C05480=1150.541,191.261,-61.437,-178.171,7.215,148.820
C05481=1150.545,191.011,-61.414,-178.174,7.213,148.820
C05482=1150.550,190.763,-61.390,-178.176,7.211,148.820
C05483=1150.554,190.514,-61.366,-178.180,7.208,148.820
C05484=1150.559,190.265,-61.343,-178.182,7.206,148.821
C05485=1150.564,190.016,-61.319,-178.185,7.203,148.821
C05486=1150.568,189.768,-61.295,-178.187,7.201,148.821
C05487=1150.573,189.519,-61.272,-178.191,7.199,148.821
C05488=1150.578,189.270,-61.249,-178.193,7.197,148.822
C05489=1150.582,189.020,-61.225,-178.196,7.194,148.822
C05490=1150.587,188.771,-61.202,-178.199,7.192,148.822
C05491=1150.591,188.523,-61.178,-178.202,7.189,148.822
C05492=1150.596,188.274,-61.155,-178.204,7.188,148.823
C05493=1150.601,188.025,-61.131,-178.208,7.185,148.823
C05494=1150.605,187.776,-61.108,-178.210,7.183,148.823
C05495=1150.609,187.527,-61.085,-178.213,7.181,148.823
C05496=1150.615,187.279,-61.062,-178.215,7.178,148.824
C05497=1150.619,187.030,-61.038,-178.218,7.177,148.824
C05498=1150.624,186.781,-61.015,-178.221,7.174,148.824
C05499=1150.628,186.532,-60.991,-178.224,7.172,148.824
C05500=1150.633,186.283,-60.968,-178.227,7.169,148.825
C05501=1150.637,186.035,-60.945,-178.229,7.167,148.825
C05502=1150.642,185.786,-60.922,-178.232,7.165,148.825
C05503=1150.647,185.537,-60.898,-178.235,7.163,148.826
C05504=1150.651,185.288,-60.875,-178.238,7.160,148.826
C05505=1150.656,185.039,-60.852,-178.240,7.158,148.826
C05506=1150.660,184.790,-60.829,-178.243,7.157,148.826
C05507=1150.665,184.541,-60.806,-178.246,7.154,148.827
C05508=1150.670,184.292,-60.783,-178.249,7.152,148.827
C05509=1150.675,184.023,-60.758,-178.252,7.149,148.827
C05510=1150.680,183.753,-60.733,-178.255,7.147,148.827
C05511=1150.684,183.483,-60.707,-178.257,7.145,148.828
C05512=1150.690,183.214,-60.682,-178.261,7.142,148.828
C05513=1150.694,182.965,-60.659,-178.264,7.140,148.828
C05514=1150.699,182.717,-60.636,-178.266,7.138,148.829
C05515=1150.704,182.467,-60.614,-178.269,7.136,148.829
C05516=1150.708,182.218,-60.590,-178.272,7.133,148.829
C05517=1150.712,181.969,-60.567,-178.274,7.131,148.829
C05518=1150.717,181.720,-60.544,-178.278,7.129,148.830
C05519=1150.722,181.471,-60.521,-178.280,7.127,148.830
C05520=1150.726,181.223,-60.498,-178.283,7.125,148.830
C05521=1150.731,180.973,-60.476,-178.286,7.122,148.831
C05522=1150.736,180.724,-60.452,-178.288,7.120,148.831
C05523=1150.740,180.476,-60.430,-178.291,7.118,148.831
C05524=1150.745,180.227,-60.406,-178.294,7.116,148.831
C05525=1150.749,179.979,-60.384,-178.297,7.113,148.832
C05526=1150.754,179.729,-60.361,-178.300,7.111,148.832
C05527=1150.759,179.480,-60.338,-178.302,7.109,148.832
C05528=1150.763,179.231,-60.315,-178.306,7.107,148.833
C05529=1150.768,178.983,-60.292,-178.308,7.105,148.833
C05530=1150.773,178.734,-60.270,-178.310,7.103,148.833
C05531=1150.777,178.484,-60.247,-178.314,7.101,148.833
C05532=1150.782,178.235,-60.223,-178.316,7.098,148.834
C05533=1150.787,177.987,-60.202,-178.319,7.096,148.834
C05534=1150.792,177.738,-60.178,-178.322,7.094,148.834
C05535=1150.796,177.489,-60.155,-178.324,7.092,148.834
C05536=1150.801,177.239,-60.133,-178.327,7.089,148.835
C05537=1150.805,176.991,-60.110,-178.330,7.088,148.835
C05538=1150.810,176.742,-60.087,-178.333,7.085,148.835
C05539=1150.814,176.493,-60.065,-178.336,7.083,148.836
C05540=1150.819,176.244,-60.042,-178.338,7.081,148.836
C05541=1150.824,175.995,-60.020,-178.342,7.079,148.836
C05542=1150.828,175.746,-59.997,-178.344,7.077,148.837
C05543=1150.833,175.497,-59.975,-178.346,7.075,148.837
C05544=1150.838,175.249,-59.952,-178.350,7.072,148.837
C05545=1150.842,174.999,-59.930,-178.352,7.070,148.837
C05546=1150.847,174.750,-59.906,-178.355,7.069,148.838
C05547=1150.852,174.502,-59.884,-178.358,7.066,148.838
C05548=1150.856,174.253,-59.862,-178.361,7.064,148.838
C05549=1150.861,174.003,-59.839,-178.363,7.061,148.839
C05550=1150.865,173.755,-59.817,-178.366,7.060,148.839
C05551=1150.870,173.506,-59.794,-178.369,7.058,148.839
C05552=1150.874,173.257,-59.771,-178.372,7.055,148.839
C05553=1150.880,173.008,-59.749,-178.374,7.053,148.840
C05554=1150.884,172.759,-59.726,-178.377,7.052,148.840
C05555=1150.889,172.511,-59.705,-178.380,7.049,148.841
C05556=1150.894,172.261,-59.682,-178.383,7.047,148.841
C05557=1150.898,172.012,-59.659,-178.385,7.045,148.841
C05558=1150.902,171.764,-59.637,-178.389,7.043,148.841
C05559=1150.907,171.515,-59.614,-178.391,7.041,148.842
C05560=1150.911,171.265,-59.592,-178.393,7.039,148.842
C05561=1150.916,171.017,-59.570,-178.397,7.036,148.842
C05562=1150.921,170.767,-59.547,-178.399,7.035,148.843
C05563=1150.926,170.519,-59.525,-178.402,7.033,148.843
C05564=1150.930,170.270,-59.503,-178.405,7.030,148.843
C05565=1150.936,170.021,-59.481,-178.408,7.028,148.843
C05566=1150.940,169.772,-59.458,-178.410,7.026,148.844
C05567=1150.944,169.522,-59.436,-178.414,7.024,148.844
C05568=1150.950,169.274,-59.414,-178.416,7.022,148.844
C05569=1150.954,169.024,-59.392,-178.419,7.020,148.845
C05570=1150.958,168.776,-59.369,-178.422,7.017,148.845
C05571=1150.963,168.527,-59.347,-178.425,7.016,148.845
C05572=1150.968,168.278,-59.325,-178.427,7.014,148.846
C05573=1150.973,168.029,-59.303,-178.430,7.011,148.846
C05574=1150.977,167.780,-59.281,-178.433,7.009,148.846
C05575=1150.981,167.531,-59.259,-178.435,7.008,148.847
C05576=1150.987,167.282,-59.236,-178.438,7.006,148.847
C05577=1150.991,167.033,-59.214,-178.441,7.003,148.847
C05578=1150.996,166.784,-59.192,-178.444,7.001,148.848
C05579=1151.000,166.535,-59.171,-178.446,7.000,148.848
C05580=1151.005,166.286,-59.149,-178.450,6.997,148.848
C05581=1151.010,166.037,-59.126,-178.452,6.995,148.848
C05582=1151.015,165.788,-59.105,-178.455,6.993,148.849
C05583=1151.019,165.539,-59.082,-178.457,6.991,148.849
C05584=1151.024,165.291,-59.060,-178.461,6.989,148.850
C05585=1151.028,165.041,-59.038,-178.463,6.987,148.850
C05586=1151.033,164.793,-59.016,-178.465,6.985,148.850
C05587=1151.037,164.543,-58.994,-178.469,6.983,148.850
C05588=1151.043,164.294,-58.972,-178.471,6.981,148.851
C05589=1151.047,164.045,-58.950,-178.474,6.979,148.851
C05590=1151.052,163.796,-58.928,-178.477,6.977,148.852
C05591=1151.056,163.547,-58.906,-178.480,6.974,148.852
C05592=1151.061,163.298,-58.885,-178.482,6.973,148.852
C05593=1151.066,163.049,-58.863,-178.485,6.971,148.852
C05594=1151.070,162.800,-58.841,-178.488,6.968,148.853
C05595=1151.075,162.551,-58.819,-178.491,6.967,148.853
C05596=1151.080,162.302,-58.798,-178.493,6.965,148.853
C05597=1151.085,162.053,-58.776,-178.496,6.963,148.854
C05598=1151.089,161.804,-58.754,-178.499,6.960,148.854
C05599=1151.094,161.555,-58.732,-178.502,6.959,148.854
C05600=1151.098,161.306,-58.710,-178.505,6.957,148.855
C05601=1151.103,161.057,-58.689,-178.507,6.955,148.855
C05602=1151.108,160.809,-58.667,-178.510,6.952,148.855
C05603=1151.112,160.559,-58.645,-178.513,6.951,148.856
C05604=1151.117,160.310,-58.624,-178.516,6.949,148.856
C05605=1151.122,160.061,-58.602,-178.518,6.947,148.856
C05606=1151.126,159.812,-58.580,-178.522,6.945,148.857
C05607=1151.131,159.563,-58.559,-178.524,6.943,148.857
C05608=1151.136,159.314,-58.537,-178.526,6.941,148.857
C05609=1151.141,159.065,-58.516,-178.529,6.939,148.858
C05610=1151.146,158.816,-58.494,-178.532,6.936,148.858
C05611=1151.150,158.567,-58.472,-178.535,6.935,148.858
C05612=1151.155,158.318,-58.450,-178.538,6.933,148.859
C05613=1151.160,158.049,-58.427,-178.541,6.930,148.859
C05614=1151.165,157.780,-58.404,-178.544,6.929,148.860
C05615=1151.170,157.511,-58.381,-178.547,6.926,148.860
C05616=1151.175,157.242,-58.357,-178.550,6.924,148.860
C05617=1151.180,156.993,-58.336,-178.553,6.923,148.861
C05618=1151.185,156.744,-58.315,-178.555,6.921,148.861
C05619=1151.189,156.495,-58.293,-178.558,6.918,148.861
C05620=1151.194,156.246,-58.272,-178.561,6.916,148.862
C05621=1151.199,155.997,-58.250,-178.563,6.915,148.862
C05622=1151.203,155.748,-58.228,-178.566,6.913,148.862
C05623=1151.208,155.498,-58.207,-178.569,6.910,148.863
C05624=1151.213,155.250,-58.186,-178.572,6.909,148.863
C05625=1151.218,155.001,-58.165,-178.575,6.907,148.863
C05626=1151.222,154.752,-58.143,-178.577,6.905,148.864
C05627=1151.226,154.503,-58.122,-178.580,6.903,148.864
C05628=1151.232,154.254,-58.101,-178.583,6.901,148.864
C05629=1151.236,154.005,-58.079,-178.586,6.899,148.865
C05630=1151.241,153.755,-58.058,-178.589,6.897,148.865
C05631=1151.245,153.507,-58.037,-178.591,6.895,148.865
C05632=1151.250,153.257,-58.016,-178.594,6.894,148.866
C05633=1151.255,153.009,-57.994,-178.597,6.891,148.866
C05634=1151.260,152.759,-57.973,-178.600,6.889,148.867
C05635=1151.264,152.511,-57.952,-178.602,6.887,148.867
C05636=1151.269,152.261,-57.931,-178.605,6.886,148.867
C05637=1151.274,152.012,-57.910,-178.608,6.884,148.868
C05638=1151.279,151.763,-57.888,-178.611,6.881,148.868
C05639=1151.283,151.514,-57.867,-178.614,6.880,148.868
C05640=1151.288,151.265,-57.846,-178.616,6.878,148.869
C05641=1151.293,151.016,-57.825,-178.619,6.876,148.869
C05642=1151.298,150.767,-57.804,-178.622,6.874,148.869
C05643=1151.302,150.518,-57.782,-178.624,6.873,148.870
C05644=1151.307,150.268,-57.761,-178.628,6.870,148.870
C05645=1151.312,150.019,-57.740,-178.630,6.868,148.870
C05646=1151.316,149.771,-57.719,-178.633,6.866,148.871
C05647=1151.321,149.521,-57.698,-178.635,6.865,148.871
C05648=1151.327,149.272,-57.677,-178.638,6.863,148.871
C05649=1151.331,149.024,-57.656,-178.641,6.861,148.872
C05650=1151.335,148.774,-57.635,-178.644,6.859,148.872
C05651=1151.340,148.525,-57.614,-178.647,6.857,148.873
C05652=1151.345,148.276,-57.593,-178.649,6.855,148.873
C05653=1151.350,148.027,-57.572,-178.652,6.854,148.873
C05654=1151.354,147.778,-57.551,-178.655,6.852,148.874
C05655=1151.359,147.529,-57.530,-178.658,6.850,148.874
C05656=1151.364,147.280,-57.510,-178.661,6.848,148.875
C05657=1151.368,147.031,-57.488,-178.664,6.846,148.875
C05658=1151.373,146.781,-57.467,-178.666,6.844,148.875
C05659=1151.378,146.532,-57.447,-178.668,6.842,148.875
C05660=1151.383,146.283,-57.426,-178.671,6.840,148.876
C05661=1151.387,146.034,-57.405,-178.674,6.839,148.876
C05662=1151.392,145.785,-57.384,-178.677,6.837,148.877
C05663=1151.397,145.537,-57.363,-178.680,6.834,148.877
C05664=1151.402,145.287,-57.342,-178.683,6.833,148.877
C05665=1151.406,145.038,-57.322,-178.685,6.831,148.878
C05666=1151.411,144.789,-57.301,-178.688,6.829,148.878
C05667=1151.416,144.540,-57.281,-178.691,6.827,148.879
C05668=1151.421,144.291,-57.260,-178.693,6.826,148.879
C05669=1151.425,144.041,-57.239,-178.696,6.824,148.879
C05670=1151.430,143.792,-57.218,-178.699,6.822,148.880
C05671=1151.434,143.543,-57.198,-178.702,6.820,148.880
C05672=1151.440,143.294,-57.177,-178.705,6.818,148.880
C05673=1151.444,143.045,-57.156,-178.708,6.816,148.881
C05674=1151.449,142.796,-57.134,-178.710,6.815,148.881
C05675=1151.453,142.547,-57.114,-178.713,6.813,148.882
C05676=1151.458,142.298,-57.094,-178.716,6.811,148.882
C05677=1151.463,142.048,-57.073,-178.718,6.809,148.882
C05678=1151.468,141.799,-57.053,-178.721,6.808,148.883
C05679=1151.473,141.550,-57.032,-178.723,6.806,148.883
C05680=1151.477,141.301,-57.012,-178.727,6.803,148.883
C05681=1151.482,141.052,-56.991,-178.729,6.801,148.884
C05682=1151.487,140.803,-56.970,-178.732,6.800,148.884
C05683=1151.491,140.554,-56.950,-178.735,6.798,148.884
C05684=1151.496,140.305,-56.930,-178.737,6.796,148.885
C05685=1151.501,140.056,-56.909,-178.740,6.795,148.885
C05686=1151.505,139.807,-56.888,-178.743,6.793,148.886
C05687=1151.511,139.558,-56.867,-178.746,6.791,148.886
C05688=1151.515,139.309,-56.847,-178.748,6.789,148.886
C05689=1151.520,139.059,-56.827,-178.751,6.788,148.887
C05690=1151.525,138.810,-56.806,-178.754,6.785,148.887
C05691=1151.529,138.561,-56.786,-178.757,6.783,148.888
C05692=1151.534,138.312,-56.766,-178.760,6.782,148.888
C05693=1151.539,138.064,-56.746,-178.762,6.780,148.888
C05694=1151.544,137.814,-56.725,-178.765,6.778,148.889
C05695=1151.549,137.565,-56.705,-178.768,6.777,148.889
C05696=1151.553,137.316,-56.685,-178.771,6.775,148.890
C05697=1151.558,137.067,-56.664,-178.773,6.773,148.890
C05698=1151.563,136.817,-56.644,-178.776,6.771,148.890
C05699=1151.568,136.568,-56.624,-178.779,6.770,148.891
C05700=1151.572,136.319,-56.603,-178.781,6.768,148.891
C05701=1151.577,136.070,-56.582,-178.784,6.766,148.891
C05702=1151.582,135.820,-56.563,-178.787,6.765,148.892
C05703=1151.586,135.571,-56.542,-178.790,6.763,148.892
C05704=1151.591,135.323,-56.522,-178.793,6.760,148.893
C05705=1151.596,135.074,-56.503,-178.796,6.759,148.893
C05706=1151.601,134.824,-56.482,-178.798,6.757,148.893
C05707=1151.606,134.575,-56.461,-178.801,6.755,148.894
C05708=1151.611,134.326,-56.442,-178.804,6.753,148.894
C05709=1151.615,134.077,-56.421,-178.806,6.752,148.895
C05710=1151.620,133.827,-56.402,-178.809,6.750,148.895
C05711=1151.624,133.578,-56.381,-178.812,6.748,148.895
C05712=1151.630,133.330,-56.361,-178.815,6.747,148.896
C05713=1151.635,133.080,-56.341,-178.818,6.745,148.896
C05714=1151.639,132.831,-56.321,-178.821,6.744,148.897
C05715=1151.644,132.582,-56.301,-178.823,6.742,148.897
C05716=1151.648,132.333,-56.281,-178.826,6.740,148.898
C05717=1151.654,132.064,-56.259,-178.829,6.738,148.898
C05718=1151.659,131.796,-56.237,-178.832,6.736,148.898
C05719=1151.664,131.527,-56.215,-178.835,6.734,148.899
C05720=1151.669,131.258,-56.194,-178.837,6.732,148.899
C05721=1151.674,131.010,-56.174,-178.840,6.731,148.900
C05722=1151.679,130.760,-56.155,-178.843,6.729,148.900
C05723=1151.683,130.511,-56.134,-178.846,6.728,148.901
C05724=1151.688,130.262,-56.115,-178.849,6.726,148.901
C05725=1151.693,130.012,-56.095,-178.851,6.724,148.901
C05726=1151.698,129.764,-56.075,-178.854,6.723,148.902
C05727=1151.703,129.514,-56.055,-178.857,6.721,148.902
C05728=1151.707,129.266,-56.035,-178.860,6.719,148.903
C05729=1151.712,129.016,-56.015,-178.862,6.717,148.903
C05730=1151.717,128.767,-55.996,-178.865,6.716,148.903
C05731=1151.722,128.518,-55.975,-178.868,6.714,148.904
C05732=1151.727,128.268,-55.955,-178.870,6.712,148.904
C05733=1151.731,128.019,-55.935,-178.873,6.711,148.904
C05734=1151.736,127.771,-55.916,-178.876,6.709,148.905
C05735=1151.741,127.521,-55.897,-178.879,6.707,148.905
C05736=1151.745,127.272,-55.876,-178.881,6.705,148.906
C05737=1151.751,127.023,-55.857,-178.884,6.704,148.906
C05738=1151.755,126.774,-55.837,-178.887,6.702,148.906
C05739=1151.760,126.524,-55.818,-178.889,6.700,148.907
C05740=1151.765,126.275,-55.797,-178.893,6.699,148.908
C05741=1151.770,126.026,-55.778,-178.895,6.697,148.908
C05742=1151.775,125.777,-55.758,-178.898,6.696,148.908
C05743=1151.779,125.527,-55.739,-178.901,6.694,148.909
C05744=1151.784,125.279,-55.719,-178.904,6.692,148.909
C05745=1151.789,125.029,-55.699,-178.906,6.690,148.909
C05746=1151.794,124.780,-55.679,-178.909,6.689,148.910
C05747=1151.799,124.531,-55.660,-178.912,6.687,148.910
C05748=1151.803,124.282,-55.641,-178.914,6.685,148.911
C05749=1151.808,124.033,-55.621,-178.917,6.684,148.911
C05750=1151.812,123.783,-55.601,-178.920,6.682,148.911
C05751=1151.818,123.534,-55.582,-178.923,6.680,148.912
C05752=1151.822,123.285,-55.562,-178.926,6.679,148.913
C05753=1151.828,123.036,-55.543,-178.928,6.677,148.913
C05754=1151.832,122.787,-55.524,-178.931,6.675,148.913
C05755=1151.837,122.537,-55.504,-178.934,6.674,148.914
C05756=1151.842,122.289,-55.484,-178.937,6.672,148.914
C05757=1151.846,122.039,-55.464,-178.939,6.670,148.915
C05758=1151.851,121.790,-55.445,-178.942,6.669,148.915
C05759=1151.856,121.541,-55.425,-178.945,6.667,148.915
C05760=1151.860,121.292,-55.406,-178.947,6.665,148.916
C05761=1151.866,121.043,-55.387,-178.950,6.663,148.916
C05762=1151.871,120.793,-55.367,-178.953,6.662,148.917
C05763=1151.875,120.544,-55.348,-178.956,6.660,148.917
C05764=1151.880,120.295,-55.329,-178.959,6.659,148.918
C05765=1151.885,120.045,-55.309,-178.962,6.657,148.918
C05766=1151.890,119.797,-55.290,-178.964,6.655,148.918
C05767=1151.895,119.547,-55.270,-178.967,6.654,148.919
C05768=1151.899,119.298,-55.251,-178.969,6.653,148.919
C05769=1151.904,119.049,-55.232,-178.972,6.651,148.920
C05770=1151.909,118.799,-55.212,-178.975,6.649,148.920
C05771=1151.913,118.551,-55.194,-178.978,6.648,148.921
C05772=1151.918,118.301,-55.174,-178.980,6.646,148.921
C05773=1151.923,118.052,-55.155,-178.983,6.645,148.921
C05774=1151.929,117.802,-55.136,-178.986,6.643,148.922
C05775=1151.933,117.554,-55.117,-178.989,6.641,148.922
C05776=1151.938,117.304,-55.098,-178.991,6.639,148.923
C05777=1151.943,117.055,-55.078,-178.994,6.638,148.923
C05778=1151.947,116.806,-55.059,-178.997,6.636,148.923
C05779=1151.952,116.556,-55.040,-179.000,6.635,148.924
C05780=1151.957,116.307,-55.020,-179.003,6.633,148.924
C05781=1151.962,116.058,-55.002,-179.005,6.631,148.925
C05782=1151.967,115.809,-54.983,-179.008,6.630,148.925
C05783=1151.971,115.559,-54.964,-179.010,6.629,148.926
C05784=1151.976,115.311,-54.944,-179.013,6.627,148.926
C05785=1151.981,115.061,-54.925,-179.016,6.625,148.926
C05786=1151.986,114.812,-54.907,-179.018,6.624,148.927
C05787=1151.991,114.563,-54.887,-179.022,6.622,148.927
C05788=1151.995,114.314,-54.868,-179.024,6.621,148.928
C05789=1152.001,114.065,-54.849,-179.027,6.619,148.928
C05790=1152.006,113.815,-54.830,-179.030,6.617,148.929
C05791=1152.010,113.566,-54.811,-179.033,6.615,148.929
C05792=1152.015,113.317,-54.792,-179.035,6.615,148.930
C05793=1152.020,113.067,-54.774,-179.038,6.613,148.930
C05794=1152.025,112.818,-54.754,-179.041,6.612,148.931
C05795=1152.029,112.569,-54.735,-179.043,6.610,148.931
C05796=1152.034,112.319,-54.716,-179.046,6.608,148.931
C05797=1152.039,112.071,-54.698,-179.049,6.606,148.932
C05798=1152.044,111.822,-54.678,-179.052,6.605,148.932
C05799=1152.049,111.572,-54.660,-179.054,6.603,148.933
C05800=1152.054,111.323,-54.641,-179.057,6.602,148.933
C05801=1152.058,111.074,-54.622,-179.060,6.601,148.934
C05802=1152.064,110.824,-54.603,-179.062,6.599,148.934
C05803=1152.068,110.576,-54.584,-179.065,6.597,148.934
C05804=1152.073,110.325,-54.566,-179.068,6.596,148.935
C05805=1152.078,110.077,-54.547,-179.070,6.594,148.935
C05806=1152.083,109.827,-54.528,-179.074,6.593,148.936
C05807=1152.088,109.578,-54.509,-179.076,6.591,148.936
C05808=1152.093,109.329,-54.491,-179.079,6.589,148.937
C05809=1152.097,109.079,-54.472,-179.081,6.588,148.937
C05810=1152.102,108.831,-54.453,-179.084,6.587,148.938
C05811=1152.107,108.581,-54.434,-179.087,6.585,148.938
C05812=1152.112,108.331,-54.416,-179.090,6.584,148.939
C05813=1152.117,108.083,-54.397,-179.093,6.582,148.939
C05814=1152.121,107.833,-54.378,-179.095,6.580,148.939
C05815=1152.126,107.584,-54.360,-179.098,6.579,148.940
C05816=1152.132,107.335,-54.341,-179.100,6.578,148.940
C05817=1152.136,107.085,-54.322,-179.103,6.576,148.941
C05818=1152.141,106.836,-54.303,-179.106,6.575,148.941
C05819=1152.146,106.587,-54.285,-179.109,6.573,148.942
C05820=1152.150,106.337,-54.266,-179.112,6.571,148.942
C05821=1152.156,106.069,-54.246,-179.114,6.570,148.943
C05822=1152.161,105.801,-54.226,-179.118,6.568,148.943
C05823=1152.167,105.533,-54.206,-179.120,6.567,148.944
C05824=1152.171,105.264,-54.186,-179.123,6.565,148.944
C05825=1152.176,105.015,-54.168,-179.126,6.564,148.945
C05826=1152.181,104.766,-54.149,-179.129,6.562,148.945
C05827=1152.186,104.517,-54.131,-179.132,6.560,148.945
C05828=1152.191,104.267,-54.113,-179.134,6.559,148.946
C05829=1152.196,104.018,-54.094,-179.137,6.558,148.946
C05830=1152.201,103.769,-54.076,-179.140,6.556,148.947
C05831=1152.205,103.519,-54.057,-179.142,6.555,148.947
C05832=1152.210,103.270,-54.039,-179.145,6.553,148.948
C05833=1152.215,103.021,-54.020,-179.147,6.552,148.948
C05834=1152.220,102.772,-54.002,-179.151,6.551,148.949
C05835=1152.225,102.522,-53.984,-179.153,6.549,148.949
C05836=1152.229,102.273,-53.965,-179.156,6.547,148.950
C05837=1152.235,102.024,-53.946,-179.159,6.546,148.950
C05838=1152.240,101.774,-53.928,-179.161,6.544,148.950
C05839=1152.245,101.525,-53.910,-179.164,6.543,148.951
C05840=1152.249,101.275,-53.892,-179.167,6.542,148.951
C05841=1152.254,101.027,-53.873,-179.170,6.540,148.952
C05842=1152.259,100.777,-53.855,-179.172,6.538,148.952
C05843=1152.264,100.528,-53.837,-179.175,6.537,148.953
C05844=1152.269,100.278,-53.818,-179.178,6.536,148.953
C05845=1152.273,100.029,-53.800,-179.180,6.534,148.954
C05846=1152.278,99.780,-53.783,-179.183,6.533,148.954
C05847=1152.283,99.531,-53.765,-179.186,6.531,148.955
C05848=1152.289,99.282,-53.745,-179.189,6.530,148.955
C05849=1152.293,99.032,-53.727,-179.191,6.529,148.956
C05850=1152.298,98.783,-53.709,-179.194,6.527,148.956
C05851=1152.303,98.534,-53.691,-179.197,6.525,148.956
C05852=1152.308,98.285,-53.673,-179.200,6.524,148.957
C05853=1152.313,98.035,-53.655,-179.203,6.522,148.958
C05854=1152.318,97.786,-53.637,-179.205,6.522,148.958
C05855=1152.322,97.536,-53.619,-179.207,6.520,148.958
C05856=1152.327,97.287,-53.601,-179.210,6.518,148.959
C05857=1152.332,97.038,-53.582,-179.213,6.517,148.959
C05858=1152.337,96.788,-53.564,-179.215,6.516,148.960
C05859=1152.342,96.539,-53.546,-179.218,6.514,148.960
C05860=1152.347,96.290,-53.528,-179.221,6.513,148.961
C05861=1152.352,96.041,-53.510,-179.224,6.511,148.961
C05862=1152.356,95.791,-53.492,-179.226,6.510,148.962
C05863=1152.361,95.542,-53.474,-179.229,6.509,148.962
C05864=1152.366,95.293,-53.456,-179.232,6.507,148.963
C05865=1152.371,95.044,-53.438,-179.235,6.506,148.963
C05866=1152.376,94.794,-53.420,-179.238,6.504,148.964
C05867=1152.381,94.545,-53.402,-179.240,6.503,148.964
C05868=1152.386,94.295,-53.385,-179.243,6.501,148.964
C05869=1152.391,94.046,-53.367,-179.246,6.500,148.965
C05870=1152.396,93.797,-53.349,-179.249,6.498,148.966
C05871=1152.401,93.548,-53.331,-179.251,6.498,148.966
C05872=1152.405,93.298,-53.312,-179.253,6.496,148.966
C05873=1152.410,93.049,-53.294,-179.257,6.495,148.967
C05874=1152.415,92.800,-53.276,-179.259,6.493,148.967
C05875=1152.420,92.550,-53.259,-179.261,6.492,148.968
C05876=1152.425,92.301,-53.241,-179.264,6.490,148.968
C05877=1152.430,92.051,-53.223,-179.267,6.489,148.969
C05878=1152.435,91.802,-53.205,-179.270,6.487,148.969
C05879=1152.439,91.553,-53.188,-179.272,6.486,148.970
C05880=1152.444,91.304,-53.171,-179.275,6.485,148.970
C05881=1152.449,91.054,-53.153,-179.278,6.483,148.971
C05882=1152.454,90.805,-53.135,-179.280,6.483,148.971
C05883=1152.459,90.556,-53.117,-179.283,6.481,148.972
C05884=1152.464,90.306,-53.099,-179.286,6.480,148.972
C05885=1152.469,90.057,-53.081,-179.289,6.478,148.973
C05886=1152.474,89.808,-53.063,-179.291,6.477,148.973
C05887=1152.479,89.559,-53.045,-179.294,6.475,148.974
C05888=1152.484,89.309,-53.029,-179.297,6.474,148.974
C05889=1152.488,89.060,-53.011,-179.300,6.472,148.975
C05890=1152.493,88.811,-52.993,-179.302,6.471,148.975
C05891=1152.499,88.561,-52.976,-179.305,6.470,148.975
C05892=1152.503,88.312,-52.958,-179.308,6.468,148.976
C05893=1152.508,88.063,-52.940,-179.310,6.468,148.977
C05894=1152.513,87.813,-52.923,-179.313,6.466,148.977
C05895=1152.518,87.564,-52.905,-179.316,6.465,148.978
C05896=1152.523,87.314,-52.888,-179.319,6.463,148.978
C05897=1152.528,87.065,-52.870,-179.321,6.462,148.978
C05898=1152.533,86.816,-52.852,-179.324,6.460,148.979
C05899=1152.537,86.567,-52.835,-179.327,6.459,148.980
C05900=1152.542,86.317,-52.817,-179.329,6.458,148.980
C05901=1152.547,86.068,-52.800,-179.332,6.456,148.980
C05902=1152.552,85.818,-52.782,-179.335,6.455,148.981
C05903=1152.557,85.569,-52.765,-179.337,6.454,148.981
C05904=1152.562,85.320,-52.747,-179.340,6.453,148.982
C05905=1152.567,85.070,-52.730,-179.343,6.451,148.982
C05906=1152.572,84.821,-52.712,-179.346,6.450,148.983
C05907=1152.577,84.572,-52.696,-179.348,6.449,148.983
C05908=1152.582,84.323,-52.678,-179.351,6.447,148.984
C05909=1152.587,84.073,-52.660,-179.354,6.446,148.984
C05910=1152.591,83.824,-52.643,-179.356,6.445,148.985
C05911=1152.596,83.574,-52.626,-179.359,6.443,148.985
C05912=1152.601,83.325,-52.608,-179.362,6.442,148.986
C05913=1152.606,83.076,-52.591,-179.364,6.441,148.986
C05914=1152.611,82.826,-52.573,-179.367,6.439,148.987
C05915=1152.616,82.577,-52.556,-179.370,6.438,148.987
C05916=1152.621,82.328,-52.540,-179.372,6.437,148.988
C05917=1152.626,82.079,-52.522,-179.375,6.435,148.988
C05918=1152.631,81.829,-52.504,-179.378,6.434,148.989
C05919=1152.635,81.580,-52.487,-179.380,6.433,148.989
C05920=1152.641,81.330,-52.470,-179.383,6.432,148.990
C05921=1152.646,81.080,-52.452,-179.386,6.430,148.990
C05922=1152.650,80.832,-52.435,-179.388,6.429,148.991
C05923=1152.656,80.583,-52.418,-179.391,6.428,148.991
C05924=1152.660,80.333,-52.401,-179.394,6.426,148.992
C05925=1152.666,80.064,-52.383,-179.397,6.426,148.992
C05926=1152.671,79.796,-52.363,-179.399,6.424,148.993
C05927=1152.676,79.528,-52.346,-179.403,6.423,148.993
C05928=1152.681,79.259,-52.327,-179.405,6.421,148.994
C05929=1152.687,79.009,-52.310,-179.408,6.420,148.995
C05930=1152.692,78.761,-52.293,-179.411,6.419,148.995
C05931=1152.697,78.511,-52.275,-179.413,6.417,148.995
C05932=1152.701,78.262,-52.259,-179.417,6.416,148.996
C05933=1152.706,78.012,-52.241,-179.419,6.415,148.996
C05934=1152.711,77.763,-52.225,-179.421,6.413,148.997
C05935=1152.716,77.514,-52.207,-179.424,6.411,148.997
C05936=1152.721,77.265,-52.190,-179.427,6.411,148.998
C05937=1152.726,77.015,-52.173,-179.430,6.409,148.998
C05938=1152.730,76.765,-52.157,-179.432,6.408,148.999
C05939=1152.736,76.516,-52.139,-179.435,6.407,149.000
C05940=1152.741,76.267,-52.123,-179.438,6.405,149.000
C05941=1152.746,76.018,-52.105,-179.440,6.405,149.000
C05942=1152.750,75.768,-52.088,-179.443,6.403,149.001
C05943=1152.755,75.518,-52.071,-179.446,6.402,149.001
C05944=1152.760,75.270,-52.055,-179.448,6.401,149.002
C05945=1152.766,75.020,-52.037,-179.451,6.399,149.003
C05946=1152.770,74.770,-52.021,-179.453,6.399,149.003
C05947=1152.775,74.521,-52.004,-179.456,6.397,149.003
C05948=1152.780,74.272,-51.987,-179.459,6.396,149.004
C05949=1152.786,74.022,-51.970,-179.461,6.395,149.004
C05950=1152.790,73.772,-51.953,-179.464,6.393,149.005
C05951=1152.795,73.524,-51.936,-179.467,6.393,149.006
C05952=1152.800,73.275,-51.919,-179.470,6.391,149.006
C05953=1152.805,73.025,-51.902,-179.472,6.389,149.006
C05954=1152.810,72.775,-51.885,-179.475,6.389,149.007
C05955=1152.815,72.526,-51.869,-179.478,6.387,149.008
C05956=1152.819,72.277,-51.852,-179.480,6.387,149.008
C05957=1152.825,72.027,-51.835,-179.483,6.385,149.009
C05958=1152.830,71.778,-51.819,-179.486,6.383,149.009
C05959=1152.834,71.529,-51.802,-179.488,6.383,149.010
C05960=1152.839,71.279,-51.785,-179.491,6.381,149.010
C05961=1152.845,71.030,-51.769,-179.493,6.380,149.011
C05962=1152.849,70.780,-51.752,-179.496,6.379,149.011
C05963=1152.854,70.530,-51.735,-179.499,6.377,149.012
C05964=1152.860,70.282,-51.719,-179.501,6.376,149.012
C05965=1152.864,70.032,-51.702,-179.505,6.375,149.013
C05966=1152.869,69.782,-51.685,-179.507,6.374,149.013
C05967=1152.874,69.534,-51.669,-179.509,6.372,149.014
C05968=1152.879,69.284,-51.652,-179.513,6.371,149.014
C05969=1152.884,69.034,-51.635,-179.515,6.370,149.015
C05970=1152.889,68.786,-51.618,-179.518,6.369,149.015
C05971=1152.894,68.535,-51.602,-179.520,6.368,149.016
C05972=1152.899,68.287,-51.586,-179.523,6.366,149.016
C05973=1152.904,68.037,-51.569,-179.526,6.366,149.017
C05974=1152.909,67.787,-51.552,-179.528,6.364,149.017
C05975=1152.914,67.539,-51.536,-179.531,6.363,149.018
C05976=1152.918,67.289,-51.519,-179.534,6.362,149.018
C05977=1152.924,67.039,-51.503,-179.536,6.361,149.019
C05978=1152.929,66.790,-51.486,-179.539,6.360,149.019
C05979=1152.933,66.540,-51.470,-179.542,6.358,149.020
C05980=1152.938,66.292,-51.453,-179.544,6.357,149.020
C05981=1152.944,66.041,-51.437,-179.547,6.356,149.021
C05982=1152.949,65.792,-51.420,-179.549,6.355,149.021
C05983=1152.954,65.543,-51.404,-179.552,6.354,149.022
C05984=1152.958,65.293,-51.387,-179.555,6.352,149.023
C05985=1152.963,65.044,-51.372,-179.557,6.352,149.023
C05986=1152.968,64.795,-51.355,-179.560,6.350,149.023
C05987=1152.974,64.545,-51.338,-179.563,6.349,149.024
C05988=1152.978,64.295,-51.322,-179.566,6.348,149.025
C05989=1152.984,64.047,-51.306,-179.568,6.347,149.025
C05990=1152.988,63.797,-51.289,-179.571,6.346,149.026
C05991=1152.993,63.548,-51.273,-179.573,6.345,149.026
C05992=1152.998,63.298,-51.257,-179.576,6.343,149.027
C05993=1153.003,63.049,-51.240,-179.579,6.343,149.027
C05994=1153.008,62.799,-51.224,-179.581,6.341,149.028
C05995=1153.013,62.550,-51.207,-179.585,6.340,149.028
C05996=1153.018,62.300,-51.192,-179.587,6.339,149.029
C05997=1153.023,62.051,-51.175,-179.589,6.337,149.029
C05998=1153.028,61.802,-51.159,-179.592,6.337,149.030
C05999=1153.033,61.552,-51.143,-179.595,6.335,149.030
C06000=1153.038,61.303,-51.126,-179.597,6.334,149.031
C06001=1153.043,61.053,-51.110,-179.600,6.333,149.031
C06002=1153.048,60.804,-51.094,-179.602,6.332,149.032
C06003=1153.052,60.554,-51.078,-179.606,6.331,149.032
C06004=1153.058,60.305,-51.062,-179.608,6.330,149.033
C06005=1153.063,60.056,-51.046,-179.611,6.328,149.034
C06006=1153.067,59.806,-51.030,-179.613,6.328,149.034
C06007=1153.072,59.558,-51.013,-179.616,6.326,149.034
C06008=1153.077,59.307,-50.997,-179.618,6.325,149.035
C06009=1153.083,59.058,-50.981,-179.621,6.324,149.036
C06010=1153.088,58.808,-50.965,-179.624,6.323,149.036
C06011=1153.093,58.559,-50.949,-179.627,6.322,149.037
C06012=1153.098,58.309,-50.932,-179.629,6.321,149.037
C06013=1153.103,58.060,-50.917,-179.632,6.319,149.038
C06014=1153.108,57.811,-50.900,-179.634,6.319,149.038
C06015=1153.112,57.561,-50.885,-179.637,6.317,149.039
C06016=1153.117,57.313,-50.869,-179.640,6.316,149.039
C06017=1153.122,57.062,-50.853,-179.642,6.315,149.040
C06018=1153.127,56.813,-50.837,-179.645,6.314,149.040
C06019=1153.132,56.564,-50.821,-179.648,6.313,149.041
C06020=1153.137,56.314,-50.805,-179.650,6.312,149.041
C06021=1153.143,56.065,-50.789,-179.653,6.311,149.042
C06022=1153.147,55.815,-50.773,-179.655,6.310,149.042
C06023=1153.153,55.566,-50.757,-179.658,6.308,149.043
C06024=1153.157,55.316,-50.741,-179.661,6.308,149.043
C06025=1153.162,55.067,-50.725,-179.664,6.306,149.044
C06026=1153.168,54.818,-50.709,-179.666,6.305,149.045
C06027=1153.173,54.568,-50.693,-179.669,6.304,149.045
C06028=1153.178,54.319,-50.677,-179.671,6.303,149.046
C06029=1153.183,54.050,-50.660,-179.674,6.302,149.046
C06030=1153.189,53.782,-50.643,-179.677,6.301,149.047
C06031=1153.193,53.513,-50.626,-179.680,6.300,149.047
C06032=1153.199,53.244,-50.609,-179.683,6.298,149.048
C06033=1153.204,52.995,-50.594,-179.685,6.298,149.049
C06034=1153.209,52.745,-50.578,-179.688,6.296,149.049
C06035=1153.214,52.496,-50.562,-179.690,6.295,149.049
C06036=1153.219,52.247,-50.546,-179.693,6.294,149.050
C06037=1153.224,51.997,-50.530,-179.696,6.293,149.051
C06038=1153.229,51.748,-50.515,-179.699,6.292,149.051
C06039=1153.234,51.498,-50.499,-179.701,6.291,149.052
C06040=1153.239,51.248,-50.483,-179.704,6.289,149.052
C06041=1153.244,50.999,-50.467,-179.706,6.289,149.053
C06042=1153.249,50.750,-50.451,-179.709,6.288,149.053
C06043=1153.254,50.501,-50.436,-179.712,6.287,149.054
C06044=1153.259,50.251,-50.420,-179.714,6.286,149.054
C06045=1153.264,50.001,-50.405,-179.717,6.284,149.055
C06046=1153.270,49.752,-50.389,-179.719,6.284,149.055
C06047=1153.274,49.502,-50.373,-179.722,6.282,149.056
C06048=1153.279,49.253,-50.358,-179.725,6.281,149.057
C06049=1153.284,49.004,-50.342,-179.727,6.280,149.057
C06050=1153.289,48.754,-50.326,-179.730,6.279,149.058
C06051=1153.293,48.505,-50.311,-179.732,6.278,149.058
C06052=1153.299,48.255,-50.295,-179.735,6.277,149.059
C06053=1153.304,48.006,-50.280,-179.738,6.276,149.059
C06054=1153.309,47.756,-50.264,-179.740,6.275,149.060
C06055=1153.314,47.507,-50.249,-179.743,6.274,149.060
C06056=1153.319,47.257,-50.233,-179.746,6.273,149.061
C06057=1153.324,47.008,-50.218,-179.748,6.272,149.061
C06058=1153.329,46.758,-50.202,-179.751,6.271,149.062
C06059=1153.334,46.509,-50.187,-179.753,6.270,149.062
C06060=1153.339,46.259,-50.171,-179.756,6.269,149.063
C06061=1153.344,46.010,-50.156,-179.759,6.267,149.063
C06062=1153.349,45.761,-50.141,-179.761,6.267,149.064
C06063=1153.354,45.511,-50.125,-179.764,6.265,149.065
C06064=1153.359,45.262,-50.110,-179.767,6.265,149.065
C06065=1153.364,45.012,-50.094,-179.769,6.264,149.066
C06066=1153.370,44.763,-50.079,-179.772,6.262,149.066
C06067=1153.374,44.513,-50.063,-179.774,6.262,149.067
C06068=1153.379,44.264,-50.048,-179.777,6.260,149.067
C06069=1153.384,44.014,-50.032,-179.780,6.260,149.068
C06070=1153.389,43.764,-50.018,-179.782,6.259,149.068
C06071=1153.395,43.515,-50.002,-179.785,6.258,149.069
C06072=1153.399,43.266,-49.987,-179.787,6.257,149.069
C06073=1153.404,43.016,-49.971,-179.790,6.255,149.070
C06074=1153.410,42.766,-49.956,-179.793,6.255,149.071
C06075=1153.414,42.517,-49.941,-179.795,6.254,149.071
C06076=1153.420,42.268,-49.925,-179.798,6.253,149.072
C06077=1153.425,42.018,-49.911,-179.800,6.252,149.072
C06078=1153.430,41.769,-49.895,-179.803,6.250,149.073
C06079=1153.434,41.519,-49.880,-179.806,6.250,149.073
C06080=1153.439,41.270,-49.864,-179.808,6.249,149.074
C06081=1153.445,41.020,-49.849,-179.811,6.247,149.074
C06082=1153.450,40.771,-49.834,-179.813,6.247,149.075
C06083=1153.455,40.521,-49.819,-179.816,6.245,149.075
C06084=1153.460,40.272,-49.804,-179.819,6.244,149.076
C06085=1153.465,40.023,-49.788,-179.821,6.244,149.077
C06086=1153.470,39.773,-49.774,-179.824,6.242,149.077
C06087=1153.475,39.523,-49.758,-179.827,6.242,149.078
C06088=1153.479,39.274,-49.743,-179.829,6.241,149.078
C06089=1153.485,39.024,-49.727,-179.832,6.240,149.079
C06090=1153.490,38.775,-49.713,-179.834,6.239,149.079
C06091=1153.495,38.525,-49.697,-179.837,6.237,149.080
C06092=1153.500,38.276,-49.682,-179.840,6.237,149.080
C06093=1153.506,38.026,-49.668,-179.842,6.236,149.081
C06094=1153.510,37.777,-49.653,-179.845,6.235,149.082
C06095=1153.515,37.528,-49.638,-179.847,6.234,149.082
C06096=1153.521,37.278,-49.623,-179.850,6.233,149.083
C06097=1153.525,37.029,-49.608,-179.853,6.232,149.083
C06098=1153.531,36.779,-49.592,-179.855,6.231,149.084
C06099=1153.535,36.529,-49.578,-179.857,6.230,149.084
C06100=1153.540,36.280,-49.562,-179.860,6.229,149.085
C06101=1153.545,36.031,-49.547,-179.863,6.228,149.085
C06102=1153.550,35.781,-49.533,-179.865,6.227,149.086
C06103=1153.555,35.531,-49.517,-179.868,6.226,149.086
C06104=1153.560,35.282,-49.503,-179.870,6.225,149.087
C06105=1153.566,35.032,-49.487,-179.874,6.224,149.088
C06106=1153.571,34.783,-49.473,-179.876,6.223,149.088
C06107=1153.575,34.533,-49.458,-179.878,6.223,149.089
C06108=1153.581,34.283,-49.443,-179.881,6.221,149.089
C06109=1153.586,34.034,-49.428,-179.884,6.221,149.090
C06110=1153.591,33.785,-49.412,-179.886,6.220,149.090
C06111=1153.596,33.535,-49.398,-179.889,6.219,149.091
C06112=1153.601,33.286,-49.383,-179.891,6.218,149.091
C06113=1153.606,33.036,-49.368,-179.893,6.217,149.092
C06114=1153.611,32.787,-49.353,-179.897,6.216,149.093
C06115=1153.616,32.537,-49.339,-179.899,6.215,149.093
C06116=1153.621,32.288,-49.323,-179.902,6.214,149.094
C06117=1153.626,32.038,-49.309,-179.904,6.213,149.094
C06118=1153.631,31.789,-49.295,-179.907,6.212,149.095
C06119=1153.636,31.539,-49.280,-179.909,6.211,149.095
C06120=1153.642,31.289,-49.265,-179.912,6.210,149.096
C06121=1153.646,31.040,-49.250,-179.915,6.209,149.096
C06122=1153.651,30.791,-49.236,-179.917,6.209,149.097
C06123=1153.657,30.541,-49.220,-179.920,6.207,149.098
C06124=1153.661,30.292,-49.206,-179.923,6.207,149.098
C06125=1153.666,30.042,-49.192,-179.925,6.206,149.099
C06126=1153.671,29.793,-49.177,-179.927,6.205,149.099
C06127=1153.677,29.543,-49.162,-179.930,6.204,149.100
C06128=1153.682,29.294,-49.148,-179.932,6.203,149.100
C06129=1153.687,29.045,-49.133,-179.935,6.202,149.101
C06130=1153.692,28.795,-49.119,-179.938,6.201,149.101
C06131=1153.697,28.545,-49.104,-179.940,6.200,149.102
C06132=1153.702,28.296,-49.089,-179.943,6.200,149.103
C06133=1153.707,28.027,-49.073,-179.946,6.198,149.103
C06134=1153.713,27.758,-49.058,-179.948,6.198,149.104
C06135=1153.719,27.488,-49.042,-179.951,6.196,149.104
C06136=1153.724,27.220,-49.026,-179.954,6.196,149.105
C06137=1153.729,26.970,-49.012,-179.956,6.195,149.105
C06138=1153.733,26.721,-48.997,-179.959,6.194,149.106
C06139=1153.739,26.472,-48.983,-179.961,6.193,149.107
C06140=1153.745,26.222,-48.968,-179.964,6.192,149.107
C06141=1153.750,25.972,-48.954,-179.967,6.191,149.108
C06142=1153.754,25.723,-48.939,-179.969,6.190,149.108
C06143=1153.759,25.473,-48.924,-179.972,6.189,149.109
C06144=1153.764,25.224,-48.910,-179.975,6.188,149.110
C06145=1153.769,24.974,-48.896,-179.977,6.187,149.110
C06146=1153.774,24.724,-48.882,-179.980,6.187,149.111
C06147=1153.780,24.475,-48.866,-179.982,6.186,149.111
C06148=1153.785,24.226,-48.852,-179.985,6.185,149.112
C06149=1153.790,23.976,-48.838,-179.987,6.184,149.112
C06150=1153.795,23.726,-48.824,-179.989,6.183,149.113
C06151=1153.800,23.477,-48.809,-179.992,6.183,149.113
C06152=1153.805,23.227,-48.795,-179.995,6.181,149.114
C06153=1153.810,22.978,-48.780,-179.997,6.180,149.115
C06154=1153.815,22.729,-48.766,-180.000,6.180,149.115
C06155=1153.820,22.479,-48.752,179.997,6.178,149.116
C06156=1153.825,22.229,-48.738,179.995,6.178,149.116
C06157=1153.830,21.980,-48.723,179.992,6.177,149.117
C06158=1153.835,21.730,-48.709,179.990,6.176,149.117
C06159=1153.840,21.481,-48.695,179.987,6.175,149.118
C06160=1153.845,21.231,-48.681,179.985,6.174,149.118
C06161=1153.850,20.982,-48.667,179.982,6.174,149.119
C06162=1153.855,20.732,-48.652,179.980,6.173,149.120
C06163=1153.860,20.482,-48.638,179.977,6.172,149.120
C06164=1153.867,20.233,-48.623,179.975,6.171,149.121
C06165=1153.872,19.983,-48.609,179.972,6.170,149.121
C06166=1153.876,19.733,-48.595,179.970,6.169,149.122
C06167=1153.881,19.484,-48.581,179.966,6.168,149.122
C06168=1153.886,19.234,-48.567,179.964,6.167,149.123
C06169=1153.891,18.985,-48.553,179.962,6.167,149.124
C06170=1153.896,18.736,-48.539,179.959,6.166,149.124
C06171=1153.901,18.486,-48.524,179.956,6.165,149.125
C06172=1153.906,18.236,-48.510,179.954,6.164,149.125
C06173=1153.912,17.987,-48.496,179.951,6.164,149.126
C06174=1153.917,17.737,-48.482,179.949,6.163,149.126
C06175=1153.922,17.488,-48.468,179.946,6.161,149.127
C06176=1153.926,17.238,-48.453,179.944,6.161,149.127
C06177=1153.932,16.989,-48.440,179.942,6.160,149.128
C06178=1153.937,16.739,-48.425,179.939,6.159,149.129
C06179=1153.942,16.490,-48.411,179.937,6.159,149.129
C06180=1153.948,16.241,-48.397,179.934,6.157,149.130
C06181=1153.952,15.991,-48.383,179.931,6.156,149.130
C06182=1153.958,15.741,-48.369,179.929,6.156,149.131
C06183=1153.963,15.491,-48.355,179.927,6.155,149.131
C06184=1153.967,15.242,-48.342,179.923,6.154,149.132
C06185=1153.972,14.992,-48.327,179.921,6.153,149.133
C06186=1153.977,14.743,-48.313,179.919,6.153,149.133
C06187=1153.983,14.494,-48.299,179.916,6.152,149.134
C06188=1153.988,14.244,-48.285,179.914,6.151,149.134
C06189=1153.993,13.994,-48.271,179.911,6.150,149.135
C06190=1153.999,13.745,-48.257,179.908,6.149,149.135
C06191=1154.003,13.495,-48.244,179.906,6.148,149.136
C06192=1154.008,13.246,-48.229,179.903,6.148,149.137
C06193=1154.013,12.997,-48.216,179.901,6.147,149.137
C06194=1154.019,12.746,-48.202,179.898,6.146,149.138
C06195=1154.024,12.496,-48.188,179.896,6.145,149.138
C06196=1154.029,12.247,-48.174,179.893,6.145,149.139
C06197=1154.033,11.998,-48.160,179.891,6.144,149.139
C06198=1154.039,11.748,-48.147,179.888,6.143,149.140
C06199=1154.044,11.499,-48.133,179.886,6.142,149.141
C06200=1154.049,11.249,-48.118,179.883,6.141,149.141
C06201=1154.054,10.999,-48.105,179.881,6.140,149.142
C06202=1154.059,10.750,-48.092,179.878,6.140,149.142
C06203=1154.064,10.500,-48.077,179.876,6.139,149.143
C06204=1154.070,10.251,-48.063,179.873,6.138,149.143
C06205=1154.075,10.001,-48.050,179.871,6.137,149.144
C06206=1154.079,9.752,-48.036,179.868,6.137,149.145
C06207=1154.085,9.503,-48.022,179.866,6.136,149.145
C06208=1154.090,9.252,-48.009,179.863,6.135,149.146
C06209=1154.095,9.002,-47.994,179.860,6.134,149.146
C06210=1154.100,8.753,-47.982,179.858,6.133,149.147
C06211=1154.105,8.503,-47.967,179.856,6.133,149.147
C06212=1154.111,8.254,-47.954,179.853,6.132,149.148
C06213=1154.115,8.004,-47.941,179.851,6.131,149.149
C06214=1154.121,7.755,-47.927,179.848,6.131,149.149
C06215=1154.126,7.505,-47.913,179.845,6.129,149.150
C06216=1154.131,7.255,-47.899,179.843,6.129,149.150
C06217=1154.136,7.007,-47.885,179.840,6.128,149.151
C06218=1154.141,6.756,-47.872,179.838,6.127,149.152
C06219=1154.147,6.507,-47.858,179.836,6.127,149.152
C06220=1154.151,6.257,-47.845,179.833,6.126,149.153
C06221=1154.157,6.008,-47.831,179.830,6.125,149.153
C06222=1154.162,5.758,-47.818,179.828,6.124,149.154
C06223=1154.166,5.509,-47.804,179.825,6.123,149.154
C06224=1154.172,5.259,-47.791,179.823,6.123,149.155
C06225=1154.176,5.010,-47.777,179.821,6.122,149.155
C06226=1154.182,4.760,-47.764,179.818,6.121,149.156
C06227=1154.187,4.510,-47.750,179.815,6.120,149.157
C06228=1154.192,4.261,-47.737,179.813,6.119,149.157
C06229=1154.197,4.011,-47.723,179.810,6.119,149.158
C06230=1154.203,3.762,-47.709,179.808,6.118,149.158
C06231=1154.207,3.512,-47.696,179.805,6.117,149.159
C06232=1154.213,3.263,-47.683,179.803,6.117,149.159
C06233=1154.217,3.013,-47.669,179.801,6.116,149.160
C06234=1154.223,2.764,-47.656,179.798,6.115,149.160
C06235=1154.228,2.513,-47.643,179.795,6.114,149.161
C06236=1154.233,2.264,-47.629,179.793,6.113,149.162
C06237=1154.239,1.994,-47.615,179.790,6.113,149.162
C06238=1154.244,1.725,-47.600,179.788,6.112,149.163
C06239=1154.250,1.457,-47.586,179.784,6.111,149.164
C06240=1154.255,1.187,-47.571,179.782,6.110,149.164
C06241=1154.260,0.937,-47.558,179.780,6.110,149.165
C06242=1154.266,0.688,-47.544,179.777,6.109,149.165
C06243=1154.271,0.437,-47.531,179.775,6.109,149.166
C06244=1154.276,0.189,-47.518,179.772,6.107,149.166
C06245=1154.281,-0.061,-47.504,179.769,6.107,149.167
C06246=1154.286,-0.311,-47.491,179.767,6.106,149.168
C06247=1154.292,-0.560,-47.477,179.765,6.105,149.168
C06248=1154.296,-0.810,-47.464,179.762,6.104,149.169
C06249=1154.302,-1.060,-47.451,179.760,6.104,149.169
C06250=1154.306,-1.310,-47.438,179.758,6.103,149.170
C06251=1154.312,-1.559,-47.424,179.755,6.103,149.171
C06252=1154.317,-1.809,-47.411,179.752,6.101,149.171
C06253=1154.322,-2.058,-47.398,179.749,6.101,149.172
C06254=1154.327,-2.307,-47.385,179.747,6.100,149.172
C06255=1154.332,-2.557,-47.372,179.745,6.099,149.173
C06256=1154.338,-2.807,-47.359,179.742,6.099,149.173
C06257=1154.342,-3.057,-47.346,179.740,6.098,149.174
C06258=1154.348,-3.306,-47.333,179.738,6.097,149.175
C06259=1154.353,-3.555,-47.319,179.735,6.097,149.175
C06260=1154.358,-3.805,-47.306,179.733,6.096,149.176
C06261=1154.363,-4.055,-47.293,179.730,6.095,149.176
C06262=1154.368,-4.305,-47.280,179.727,6.094,149.177
C06263=1154.374,-4.554,-47.267,179.725,6.094,149.178
C06264=1154.378,-4.803,-47.254,179.723,6.093,149.178
C06265=1154.384,-5.053,-47.240,179.720,6.092,149.179
C06266=1154.389,-5.303,-47.227,179.718,6.092,149.179
C06267=1154.394,-5.552,-47.215,179.715,6.091,149.180
C06268=1154.399,-5.802,-47.201,179.713,6.090,149.180
C06269=1154.404,-6.052,-47.189,179.710,6.090,149.181
C06270=1154.410,-6.302,-47.175,179.708,6.089,149.181
C06271=1154.414,-6.551,-47.162,179.705,6.089,149.182
C06272=1154.419,-6.800,-47.149,179.703,6.087,149.183
C06273=1154.425,-7.050,-47.136,179.700,6.087,149.183
C06274=1154.430,-7.300,-47.123,179.698,6.086,149.184
C06275=1154.435,-7.549,-47.110,179.695,6.085,149.184
C06276=1154.440,-7.799,-47.097,179.693,6.085,149.185
C06277=1154.445,-8.049,-47.084,179.690,6.084,149.186
C06278=1154.451,-8.298,-47.072,179.688,6.083,149.186
C06279=1154.455,-8.548,-47.059,179.685,6.083,149.187
C06280=1154.461,-8.798,-47.046,179.683,6.082,149.187
C06281=1154.466,-9.047,-47.033,179.681,6.082,149.188
C06282=1154.471,-9.297,-47.020,179.678,6.081,149.188
C06283=1154.476,-9.547,-47.007,179.676,6.080,149.189
C06284=1154.482,-9.796,-46.994,179.674,6.080,149.190
C06285=1154.487,-10.045,-46.982,179.670,6.078,149.190
C06286=1154.491,-10.295,-46.969,179.668,6.077,149.191
C06287=1154.497,-10.545,-46.955,179.666,6.077,149.191
C06288=1154.502,-10.794,-46.943,179.663,6.076,149.192
C06289=1154.507,-11.044,-46.930,179.661,6.076,149.193
C06290=1154.512,-11.294,-46.917,179.659,6.075,149.193
C06291=1154.518,-11.543,-46.904,179.656,6.075,149.194
C06292=1154.523,-11.793,-46.891,179.654,6.074,149.194
C06293=1154.527,-12.043,-46.878,179.651,6.073,149.195
C06294=1154.532,-12.292,-46.866,179.649,6.073,149.195
C06295=1154.538,-12.541,-46.853,179.646,6.072,149.196
C06296=1154.543,-12.791,-46.840,179.644,6.071,149.197
C06297=1154.548,-13.041,-46.828,179.641,6.071,149.197
C06298=1154.553,-13.291,-46.815,179.639,6.070,149.198
C06299=1154.558,-13.540,-46.803,179.637,6.070,149.198
C06300=1154.564,-13.790,-46.789,179.634,6.069,149.199
C06301=1154.569,-14.040,-46.776,179.632,6.068,149.200
C06302=1154.574,-14.289,-46.764,179.630,6.068,149.200
C06303=1154.579,-14.538,-46.751,179.627,6.067,149.201
C06304=1154.584,-14.788,-46.739,179.624,6.066,149.201
C06305=1154.589,-15.038,-46.726,179.621,6.065,149.202
C06306=1154.595,-15.288,-46.713,179.619,6.064,149.202
C06307=1154.600,-15.537,-46.701,179.617,6.064,149.203
C06308=1154.605,-15.787,-46.688,179.614,6.063,149.203
C06309=1154.610,-16.036,-46.675,179.612,6.063,149.204
C06310=1154.615,-16.287,-46.663,179.610,6.062,149.205
C06311=1154.620,-16.536,-46.651,179.607,6.061,149.205
C06312=1154.625,-16.785,-46.638,179.605,6.061,149.206
C06313=1154.631,-17.034,-46.625,179.602,6.060,149.207
C06314=1154.637,-17.285,-46.613,179.600,6.059,149.207
C06315=1154.641,-17.535,-46.600,179.597,6.059,149.208
C06316=1154.646,-17.784,-46.587,179.595,6.058,149.208
C06317=1154.651,-18.033,-46.575,179.592,6.058,149.209
C06318=1154.657,-18.283,-46.563,179.590,6.057,149.209
C06319=1154.662,-18.533,-46.550,179.588,6.056,149.210
C06320=1154.667,-18.782,-46.538,179.585,6.056,149.210
C06321=1154.672,-19.033,-46.525,179.583,6.055,149.211
C06322=1154.677,-19.282,-46.513,179.581,6.054,149.212
C06323=1154.682,-19.531,-46.500,179.578,6.054,149.212
C06324=1154.687,-19.781,-46.488,179.576,6.053,149.213
C06325=1154.693,-20.030,-46.476,179.573,6.053,149.214
C06326=1154.698,-20.280,-46.463,179.571,6.052,149.214
C06327=1154.703,-20.530,-46.451,179.568,6.051,149.215
C06328=1154.709,-20.779,-46.438,179.566,6.051,149.215
C06329=1154.714,-21.029,-46.425,179.563,6.050,149.216
C06330=1154.719,-21.279,-46.413,179.561,6.049,149.216
C06331=1154.724,-21.529,-46.401,179.559,6.049,149.217
C06332=1154.729,-21.778,-46.388,179.556,6.048,149.217
C06333=1154.735,-22.028,-46.376,179.554,6.048,149.218
C06334=1154.740,-22.277,-46.363,179.551,6.047,149.219
C06335=1154.745,-22.527,-46.352,179.549,6.047,149.219
C06336=1154.750,-22.776,-46.339,179.547,6.046,149.220
C06337=1154.756,-23.026,-46.326,179.544,6.045,149.220
C06338=1154.761,-23.276,-46.315,179.542,6.045,149.221
C06339=1154.766,-23.526,-46.302,179.539,6.044,149.222
C06340=1154.770,-23.775,-46.290,179.537,6.043,149.222
C06341=1154.777,-24.045,-46.276,179.534,6.043,149.223
C06342=1154.782,-24.315,-46.263,179.532,6.042,149.223
C06343=1154.787,-24.585,-46.250,179.529,6.042,149.224
C06344=1154.794,-24.855,-46.237,179.526,6.040,149.225
C06345=1154.798,-25.104,-46.225,179.525,6.040,149.225
C06346=1154.803,-25.354,-46.213,179.522,6.040,149.226
C06347=1154.809,-25.604,-46.201,179.520,6.039,149.226
C06348=1154.814,-25.853,-46.188,179.517,6.039,149.227
C06349=1154.819,-26.103,-46.176,179.515,6.038,149.228
C06350=1154.824,-26.353,-46.163,179.512,6.038,149.228
C06351=1154.829,-26.603,-46.151,179.510,6.037,149.229
C06352=1154.835,-26.853,-46.140,179.507,6.036,149.229
C06353=1154.840,-27.102,-46.127,179.505,6.036,149.230
C06354=1154.845,-27.352,-46.116,179.503,6.035,149.231
C06355=1154.850,-27.601,-46.103,179.500,6.034,149.231
C06356=1154.855,-27.851,-46.091,179.498,6.034,149.232
C06357=1154.860,-28.100,-46.079,179.496,6.033,149.232
C06358=1154.866,-28.350,-46.067,179.493,6.033,149.233
C06359=1154.871,-28.600,-46.055,179.491,6.032,149.233
C06360=1154.876,-28.849,-46.042,179.488,6.031,149.234
C06361=1154.881,-29.099,-46.031,179.486,6.031,149.235
C06362=1154.886,-29.349,-46.019,179.483,6.030,149.235
C06363=1154.891,-29.598,-46.006,179.481,6.029,149.236
C06364=1154.897,-29.848,-45.994,179.478,6.029,149.236
C06365=1154.902,-30.098,-45.982,179.476,6.028,149.237
C06366=1154.907,-30.347,-45.971,179.474,6.028,149.238
C06367=1154.912,-30.597,-45.959,179.471,6.027,149.238
C06368=1154.917,-30.846,-45.946,179.469,6.027,149.239
C06369=1154.923,-31.096,-45.934,179.466,6.026,149.239
C06370=1154.928,-31.346,-45.922,179.464,6.025,149.240
C06371=1154.933,-31.596,-45.911,179.462,6.025,149.240
C06372=1154.938,-31.845,-45.898,179.460,6.025,149.241
C06373=1154.943,-32.095,-45.887,179.457,6.024,149.242
C06374=1154.949,-32.344,-45.875,179.455,6.023,149.242
C06375=1154.954,-32.593,-45.863,179.453,6.023,149.243
C06376=1154.959,-32.843,-45.851,179.450,6.022,149.243
C06377=1154.965,-33.093,-45.839,179.448,6.022,149.244
C06378=1154.970,-33.343,-45.827,179.446,6.021,149.244
C06379=1154.975,-33.593,-45.816,179.443,6.020,149.245
C06380=1154.980,-33.842,-45.803,179.441,6.020,149.246
C06381=1154.985,-34.092,-45.792,179.438,6.019,149.246
C06382=1154.991,-34.342,-45.780,179.436,6.018,149.247
C06383=1154.995,-34.592,-45.768,179.433,6.018,149.247
C06384=1155.001,-34.841,-45.756,179.431,6.017,149.248
C06385=1155.006,-35.091,-45.744,179.429,6.018,149.249
C06386=1155.011,-35.341,-45.733,179.427,6.017,149.249
C06387=1155.016,-35.591,-45.721,179.424,6.016,149.250
C06388=1155.022,-35.840,-45.709,179.422,6.016,149.250
C06389=1155.028,-36.090,-45.697,179.419,6.015,149.251
C06390=1155.032,-36.339,-45.685,179.417,6.014,149.251
C06391=1155.037,-36.589,-45.673,179.414,6.014,149.252
C06392=1155.043,-36.839,-45.662,179.412,6.013,149.253
C06393=1155.047,-37.088,-45.650,179.410,6.013,149.253
C06394=1155.053,-37.338,-45.638,179.407,6.012,149.254
C06395=1155.058,-37.588,-45.627,179.405,6.012,149.254
C06396=1155.064,-37.837,-45.616,179.402,6.011,149.255
C06397=1155.069,-38.087,-45.604,179.400,6.011,149.256
C06398=1155.074,-38.337,-45.592,179.398,6.010,149.256
C06399=1155.079,-38.587,-45.581,179.396,6.010,149.257
C06400=1155.084,-38.836,-45.568,179.393,6.009,149.257
C06401=1155.089,-39.085,-45.557,179.391,6.008,149.258
C06402=1155.094,-39.335,-45.545,179.389,6.008,149.258
C06403=1155.100,-39.585,-45.533,179.386,6.007,149.259
C06404=1155.105,-39.834,-45.522,179.384,6.007,149.260
C06405=1155.111,-40.084,-45.510,179.381,6.006,149.260
C06406=1155.115,-40.334,-45.499,179.379,6.006,149.261
C06407=1155.121,-40.584,-45.487,179.377,6.006,149.261
C06408=1155.126,-40.834,-45.475,179.375,6.005,149.262
C06409=1155.131,-41.083,-45.464,179.372,6.004,149.262
C06410=1155.137,-41.333,-45.452,179.370,6.004,149.263
C06411=1155.142,-41.582,-45.441,179.368,6.003,149.264
C06412=1155.147,-41.832,-45.429,179.365,6.003,149.264
C06413=1155.152,-42.082,-45.418,179.363,6.002,149.265
C06414=1155.158,-42.331,-45.406,179.360,6.002,149.266
C06415=1155.162,-42.581,-45.395,179.358,6.001,149.266
C06416=1155.168,-42.831,-45.383,179.356,6.001,149.267
C06417=1155.173,-43.080,-45.372,179.354,6.000,149.267
C06418=1155.178,-43.331,-45.361,179.351,6.000,149.268
C06419=1155.184,-43.580,-45.350,179.349,5.999,149.268
C06420=1155.189,-43.830,-45.338,179.347,5.998,149.269
C06421=1155.194,-44.080,-45.326,179.344,5.998,149.270
C06422=1155.199,-44.329,-45.315,179.342,5.997,149.270
C06423=1155.204,-44.578,-45.304,179.339,5.997,149.271
C06424=1155.210,-44.828,-45.292,179.337,5.997,149.271
C06425=1155.215,-45.078,-45.281,179.335,5.996,149.272
C06426=1155.220,-45.328,-45.269,179.333,5.996,149.272
C06427=1155.225,-45.577,-45.257,179.330,5.995,149.273
C06428=1155.231,-45.827,-45.247,179.328,5.994,149.274
C06429=1155.236,-46.077,-45.235,179.325,5.994,149.274
C06430=1155.241,-46.327,-45.223,179.323,5.993,149.275
C06431=1155.246,-46.576,-45.212,179.321,5.994,149.275
C06432=1155.252,-46.825,-45.201,179.319,5.993,149.276
C06433=1155.257,-47.075,-45.189,179.316,5.992,149.276
C06434=1155.262,-47.326,-45.178,179.314,5.992,149.277
C06435=1155.268,-47.575,-45.167,179.312,5.991,149.278
C06436=1155.272,-47.824,-45.156,179.309,5.990,149.278
C06437=1155.278,-48.074,-45.144,179.307,5.990,149.279
C06438=1155.283,-48.324,-45.133,179.305,5.990,149.279
C06439=1155.289,-48.574,-45.122,179.302,5.989,149.280
C06440=1155.293,-48.823,-45.111,179.300,5.989,149.281
C06441=1155.298,-49.073,-45.099,179.298,5.988,149.281
C06442=1155.304,-49.322,-45.088,179.295,5.988,149.282
C06443=1155.309,-49.572,-45.077,179.293,5.987,149.282
C06444=1155.315,-49.822,-45.065,179.290,5.986,149.283
C06445=1155.321,-50.093,-45.053,179.288,5.986,149.283
C06446=1155.326,-50.363,-45.042,179.285,5.985,149.284
C06447=1155.331,-50.634,-45.030,179.283,5.984,149.285
C06448=1155.337,-50.904,-45.017,179.280,5.984,149.285
C06449=1155.342,-51.154,-45.006,179.278,5.984,149.286
C06450=1155.348,-51.404,-44.994,179.276,5.984,149.286
C06451=1155.353,-51.653,-44.984,179.273,5.983,149.287
C06452=1155.358,-51.903,-44.973,179.271,5.982,149.288
C06453=1155.363,-52.153,-44.961,179.269,5.982,149.288
C06454=1155.369,-52.402,-44.950,179.266,5.981,149.289
C06455=1155.374,-52.652,-44.940,179.265,5.981,149.289
C06456=1155.379,-52.902,-44.928,179.262,5.981,149.290
C06457=1155.384,-53.151,-44.917,179.260,5.980,149.291
C06458=1155.389,-53.401,-44.906,179.257,5.980,149.291
C06459=1155.395,-53.651,-44.895,179.255,5.979,149.292
C06460=1155.400,-53.901,-44.884,179.252,5.978,149.292
C06461=1155.405,-54.151,-44.873,179.251,5.978,149.293
C06462=1155.410,-54.399,-44.862,179.249,5.978,149.293
C06463=1155.416,-54.650,-44.851,179.246,5.977,149.294
C06464=1155.421,-54.900,-44.839,179.244,5.976,149.295
C06465=1155.426,-55.149,-44.829,179.241,5.976,149.295
C06466=1155.431,-55.399,-44.818,179.240,5.976,149.296
C06467=1155.437,-55.649,-44.807,179.237,5.976,149.296
C06468=1155.442,-55.898,-44.796,179.235,5.975,149.297
C06469=1155.447,-56.148,-44.785,179.232,5.974,149.298
C06470=1155.452,-56.397,-44.774,179.230,5.974,149.298
C06471=1155.458,-56.647,-44.762,179.228,5.974,149.299
C06472=1155.463,-56.898,-44.752,179.226,5.973,149.299
C06473=1155.468,-57.147,-44.741,179.223,5.972,149.300
C06474=1155.473,-57.397,-44.730,179.221,5.972,149.300
C06475=1155.478,-57.646,-44.719,179.219,5.971,149.301
C06476=1155.484,-57.896,-44.708,179.216,5.971,149.302
C06477=1155.489,-58.145,-44.697,179.214,5.971,149.302
C06478=1155.494,-58.395,-44.687,179.212,5.971,149.303
C06479=1155.499,-58.645,-44.676,179.209,5.970,149.303
C06480=1155.505,-58.895,-44.665,179.207,5.969,149.304
C06481=1155.510,-59.145,-44.653,179.205,5.969,149.304
C06482=1155.516,-59.394,-44.643,179.203,5.969,149.305
C06483=1155.521,-59.644,-44.633,179.200,5.968,149.306
C06484=1155.526,-59.893,-44.622,179.198,5.967,149.306
C06485=1155.531,-60.144,-44.611,179.195,5.967,149.307
C06486=1155.536,-60.393,-44.600,179.194,5.967,149.307
C06487=1155.541,-60.643,-44.590,179.192,5.966,149.308
C06488=1155.547,-60.893,-44.578,179.189,5.966,149.309
C06489=1155.552,-61.142,-44.568,179.187,5.965,149.309
C06490=1155.557,-61.392,-44.557,179.184,5.965,149.310
C06491=1155.563,-61.641,-44.546,179.183,5.965,149.310
C06492=1155.568,-61.892,-44.535,179.180,5.964,149.311
C06493=1155.573,-62.141,-44.525,179.178,5.963,149.311
C06494=1155.578,-62.391,-44.514,179.176,5.963,149.312
C06495=1155.583,-62.640,-44.504,179.173,5.962,149.313
C06496=1155.589,-62.890,-44.492,179.171,5.962,149.313
C06497=1155.595,-63.140,-44.482,179.169,5.962,149.314
C06498=1155.600,-63.390,-44.471,179.166,5.961,149.314
C06499=1155.605,-63.639,-44.460,179.164,5.961,149.315
C06500=1155.610,-63.889,-44.450,179.162,5.961,149.315
C06501=1155.615,-64.139,-44.439,179.160,5.960,149.316
C06502=1155.620,-64.388,-44.428,179.157,5.960,149.317
C06503=1155.626,-64.638,-44.418,179.155,5.959,149.317
C06504=1155.631,-64.888,-44.407,179.153,5.959,149.318
C06505=1155.636,-65.138,-44.397,179.151,5.958,149.318
C06506=1155.641,-65.387,-44.386,179.148,5.958,149.319
C06507=1155.647,-65.637,-44.376,179.146,5.957,149.319
C06508=1155.652,-65.887,-44.365,179.144,5.956,149.320
C06509=1155.657,-66.137,-44.355,179.142,5.957,149.321
C06510=1155.662,-66.386,-44.344,179.140,5.956,149.321
C06511=1155.667,-66.636,-44.333,179.137,5.956,149.322
C06512=1155.673,-66.885,-44.323,179.135,5.955,149.322
C06513=1155.678,-67.136,-44.313,179.133,5.955,149.323
C06514=1155.683,-67.385,-44.302,179.130,5.955,149.323
C06515=1155.688,-67.635,-44.291,179.128,5.954,149.324
C06516=1155.694,-67.884,-44.281,179.126,5.953,149.325
C06517=1155.699,-68.135,-44.270,179.124,5.953,149.325
C06518=1155.705,-68.384,-44.260,179.121,5.953,149.326
C06519=1155.710,-68.633,-44.249,179.119,5.952,149.326
C06520=1155.715,-68.883,-44.239,179.117,5.951,149.327
C06521=1155.720,-69.133,-44.228,179.115,5.952,149.328
C06522=1155.725,-69.383,-44.218,179.113,5.951,149.328
C06523=1155.731,-69.633,-44.208,179.110,5.951,149.329
C06524=1155.736,-69.883,-44.197,179.108,5.950,149.329
C06525=1155.742,-70.132,-44.187,179.106,5.950,149.330
C06526=1155.747,-70.381,-44.176,179.104,5.949,149.330
C06527=1155.752,-70.632,-44.165,179.101,5.949,149.331
C06528=1155.758,-70.881,-44.155,179.099,5.948,149.332
C06529=1155.763,-71.131,-44.145,179.097,5.948,149.332
C06530=1155.768,-71.381,-44.134,179.095,5.948,149.333
C06531=1155.774,-71.630,-44.124,179.092,5.947,149.333
C06532=1155.779,-71.881,-44.114,179.091,5.947,149.334
C06533=1155.784,-72.130,-44.103,179.088,5.947,149.334
C06534=1155.790,-72.380,-44.093,179.086,5.946,149.335
C06535=1155.794,-72.630,-44.083,179.084,5.945,149.335
C06536=1155.800,-72.879,-44.073,179.081,5.946,149.336
C06537=1155.805,-73.128,-44.062,179.079,5.945,149.337
C06538=1155.810,-73.378,-44.051,179.077,5.944,149.337
C06539=1155.816,-73.628,-44.041,179.074,5.944,149.338
C06540=1155.821,-73.877,-44.031,179.073,5.944,149.338
C06541=1155.826,-74.128,-44.020,179.070,5.943,149.339
C06542=1155.832,-74.377,-44.010,179.068,5.943,149.339
C06543=1155.837,-74.627,-44.000,179.066,5.943,149.340
C06544=1155.842,-74.877,-43.990,179.064,5.942,149.341
C06545=1155.847,-75.126,-43.980,179.062,5.941,149.341
C06546=1155.853,-75.376,-43.970,179.059,5.941,149.342
C06547=1155.858,-75.626,-43.959,179.057,5.941,149.342
C06548=1155.863,-75.876,-43.949,179.055,5.941,149.343
C06549=1155.869,-76.147,-43.938,179.052,5.940,149.343
C06550=1155.876,-76.418,-43.927,179.050,5.940,149.344
C06551=1155.881,-76.690,-43.916,179.048,5.939,149.345
C06552=1155.887,-76.961,-43.905,179.045,5.939,149.345
C06553=1155.892,-77.211,-43.895,179.043,5.938,149.346
C06554=1155.897,-77.460,-43.885,179.041,5.938,149.347
C06555=1155.902,-77.710,-43.875,179.038,5.937,149.347
C06556=1155.908,-77.960,-43.864,179.037,5.937,149.348
C06557=1155.913,-78.209,-43.854,179.034,5.937,149.348
C06558=1155.918,-78.460,-43.844,179.032,5.936,149.349
C06559=1155.923,-78.709,-43.834,179.030,5.936,149.349
C06560=1155.929,-78.958,-43.824,179.028,5.936,149.350
C06561=1155.935,-79.209,-43.814,179.025,5.935,149.350
C06562=1155.940,-79.459,-43.804,179.023,5.935,149.351
C06563=1155.945,-79.708,-43.793,179.021,5.935,149.352
C06564=1155.950,-79.958,-43.784,179.019,5.934,149.352
C06565=1155.956,-80.207,-43.774,179.016,5.933,149.353
C06566=1155.961,-80.457,-43.763,179.015,5.933,149.353
C06567=1155.966,-80.707,-43.753,179.012,5.933,149.354
C06568=1155.971,-80.957,-43.744,179.010,5.932,149.354
C06569=1155.976,-81.207,-43.733,179.008,5.932,149.355
C06570=1155.982,-81.457,-43.723,179.006,5.932,149.356
C06571=1155.987,-81.706,-43.714,179.003,5.931,149.356
C06572=1155.993,-81.955,-43.703,179.002,5.931,149.357
C06573=1155.998,-82.206,-43.694,178.999,5.931,149.357
C06574=1156.003,-82.456,-43.683,178.997,5.930,149.358
C06575=1156.008,-82.705,-43.674,178.995,5.930,149.358
C06576=1156.014,-82.955,-43.663,178.993,5.930,149.359
C06577=1156.019,-83.204,-43.653,178.990,5.929,149.359
C06578=1156.024,-83.455,-43.644,178.988,5.929,149.360
C06579=1156.030,-83.704,-43.634,178.986,5.929,149.361
C06580=1156.035,-83.954,-43.624,178.984,5.928,149.361
C06581=1156.040,-84.203,-43.614,178.982,5.928,149.362
C06582=1156.046,-84.453,-43.604,178.980,5.927,149.362
C06583=1156.051,-84.703,-43.594,178.978,5.927,149.363
C06584=1156.056,-84.953,-43.584,178.975,5.926,149.364
C06585=1156.062,-85.203,-43.575,178.973,5.926,149.364
C06586=1156.067,-85.452,-43.565,178.971,5.925,149.365
C06587=1156.072,-85.702,-43.555,178.968,5.925,149.365
C06588=1156.077,-85.952,-43.544,178.967,5.925,149.366
C06589=1156.082,-86.202,-43.535,178.964,5.925,149.366
C06590=1156.088,-86.451,-43.525,178.962,5.924,149.367
C06591=1156.094,-86.701,-43.515,178.960,5.924,149.367
C06592=1156.099,-86.951,-43.506,178.958,5.924,149.368
C06593=1156.104,-87.201,-43.496,178.956,5.924,149.369
C06594=1156.109,-87.450,-43.486,178.954,5.923,149.369
C06595=1156.115,-87.700,-43.476,178.951,5.922,149.370
C06596=1156.120,-87.950,-43.466,178.950,5.922,149.370
C06597=1156.125,-88.199,-43.457,178.947,5.922,149.371
C06598=1156.131,-88.449,-43.447,178.945,5.921,149.371
C06599=1156.135,-88.699,-43.437,178.943,5.921,149.372
C06600=1156.141,-88.949,-43.428,178.941,5.921,149.372
C06601=1156.146,-89.199,-43.418,178.938,5.920,149.373
C06602=1156.151,-89.448,-43.408,178.937,5.920,149.374
C06603=1156.157,-89.698,-43.398,178.935,5.919,149.374
C06604=1156.162,-89.947,-43.389,178.932,5.919,149.375
C06605=1156.168,-90.198,-43.379,178.930,5.919,149.375
C06606=1156.172,-90.448,-43.369,178.928,5.918,149.376
C06607=1156.178,-90.697,-43.359,178.925,5.918,149.376
C06608=1156.183,-90.947,-43.350,178.924,5.918,149.377
C06609=1156.189,-91.197,-43.340,178.922,5.917,149.377
C06610=1156.194,-91.446,-43.331,178.919,5.917,149.378
C06611=1156.200,-91.696,-43.321,178.917,5.917,149.379
C06612=1156.205,-91.946,-43.312,178.915,5.916,149.379
C06613=1156.210,-92.195,-43.302,178.913,5.917,149.380
C06614=1156.215,-92.445,-43.293,178.911,5.916,149.380
C06615=1156.220,-92.695,-43.282,178.909,5.915,149.381
C06616=1156.226,-92.945,-43.273,178.907,5.915,149.382
C06617=1156.231,-93.195,-43.263,178.904,5.915,149.382
C06618=1156.236,-93.445,-43.254,178.902,5.914,149.382
C06619=1156.242,-93.694,-43.244,178.900,5.914,149.383
C06620=1156.247,-93.944,-43.235,178.898,5.914,149.384
C06621=1156.253,-94.194,-43.225,178.896,5.913,149.384
C06622=1156.258,-94.443,-43.216,178.894,5.913,149.385
C06623=1156.264,-94.693,-43.206,178.891,5.912,149.385
C06624=1156.269,-94.943,-43.197,178.890,5.912,149.386
C06625=1156.275,-95.193,-43.187,178.887,5.912,149.387
C06626=1156.279,-95.442,-43.178,178.885,5.911,149.387
C06627=1156.285,-95.692,-43.169,178.883,5.911,149.388
C06628=1156.290,-95.942,-43.159,178.881,5.911,149.388
C06629=1156.295,-96.192,-43.149,178.879,5.910,149.389
C06630=1156.300,-96.442,-43.139,178.877,5.910,149.389
C06631=1156.306,-96.692,-43.130,178.875,5.909,149.390
C06632=1156.311,-96.942,-43.121,178.873,5.910,149.390
C06633=1156.316,-97.191,-43.111,178.871,5.909,149.391
C06634=1156.321,-97.441,-43.102,178.868,5.908,149.391
C06635=1156.327,-97.690,-43.092,178.866,5.909,149.392
C06636=1156.332,-97.940,-43.083,178.864,5.908,149.393
C06637=1156.338,-98.190,-43.074,178.862,5.908,149.393
C06638=1156.343,-98.440,-43.064,178.860,5.908,149.394
C06639=1156.348,-98.689,-43.055,178.858,5.907,149.394
C06640=1156.354,-98.940,-43.046,178.856,5.907,149.395
C06641=1156.359,-99.189,-43.036,178.854,5.906,149.395
C06642=1156.365,-99.439,-43.027,178.851,5.906,149.396
C06643=1156.370,-99.689,-43.018,178.850,5.906,149.396
C06644=1156.375,-99.938,-43.008,178.847,5.905,149.397
C06645=1156.381,-100.188,-42.999,178.845,5.905,149.398
C06646=1156.386,-100.438,-42.990,178.843,5.905,149.398
C06647=1156.391,-100.687,-42.980,178.841,5.904,149.399
C06648=1156.397,-100.937,-42.971,178.839,5.904,149.399
C06649=1156.402,-101.187,-42.962,178.837,5.904,149.400
C06650=1156.407,-101.437,-42.953,178.835,5.904,149.400
C06651=1156.413,-101.687,-42.943,178.833,5.903,149.401
C06652=1156.418,-101.937,-42.934,178.830,5.902,149.401
C06653=1156.423,-102.209,-42.924,178.829,5.903,149.402
C06654=1156.430,-102.480,-42.914,178.826,5.902,149.403
C06655=1156.435,-102.752,-42.904,178.824,5.901,149.403
C06656=1156.441,-103.025,-42.893,178.822,5.902,149.404
C06657=1156.447,-103.274,-42.884,178.819,5.901,149.404
C06658=1156.452,-103.524,-42.876,178.817,5.900,149.405
C06659=1156.457,-103.773,-42.866,178.816,5.900,149.405
C06660=1156.463,-104.024,-42.856,178.813,5.900,149.406
C06661=1156.468,-104.273,-42.848,178.811,5.900,149.407
C06662=1156.473,-104.523,-42.839,178.809,5.899,149.407
C06663=1156.478,-104.773,-42.830,178.806,5.899,149.408
C06664=1156.484,-105.023,-42.820,178.805,5.899,149.408
C06665=1156.489,-105.273,-42.811,178.803,5.898,149.409
C06666=1156.495,-105.522,-42.802,178.801,5.898,149.409
C06667=1156.500,-105.772,-42.793,178.798,5.898,149.410
C06668=1156.506,-106.022,-42.784,178.796,5.897,149.410
C06669=1156.511,-106.272,-42.775,178.795,5.897,149.411
C06670=1156.516,-106.521,-42.766,178.792,5.896,149.411
C06671=1156.521,-106.771,-42.756,178.790,5.897,149.412
C06672=1156.527,-107.021,-42.747,178.788,5.896,149.413
C06673=1156.532,-107.271,-42.738,178.787,5.896,149.413
C06674=1156.537,-107.521,-42.729,178.784,5.895,149.414
C06675=1156.542,-107.770,-42.720,178.782,5.895,149.414
C06676=1156.547,-108.020,-42.711,178.780,5.895,149.415
C06677=1156.553,-108.270,-42.702,178.778,5.894,149.415
C06678=1156.559,-108.520,-42.693,178.776,5.895,149.416
C06679=1156.564,-108.769,-42.684,178.774,5.894,149.416
C06680=1156.569,-109.019,-42.675,178.772,5.894,149.417
C06681=1156.574,-109.268,-42.666,178.770,5.893,149.417
C06682=1156.580,-109.519,-42.656,178.767,5.893,149.418
C06683=1156.585,-109.768,-42.647,178.766,5.893,149.419
C06684=1156.590,-110.018,-42.639,178.763,5.892,149.419
C06685=1156.596,-110.268,-42.630,178.762,5.892,149.420
C06686=1156.601,-110.517,-42.621,178.759,5.892,149.420
C06687=1156.607,-110.767,-42.612,178.757,5.892,149.421
C06688=1156.613,-111.017,-42.603,178.755,5.891,149.421
C06689=1156.618,-111.267,-42.594,178.754,5.891,149.422
C06690=1156.623,-111.517,-42.585,178.751,5.890,149.422
C06691=1156.628,-111.767,-42.576,178.749,5.890,149.423
C06692=1156.633,-112.017,-42.567,178.747,5.890,149.423
C06693=1156.639,-112.266,-42.559,178.745,5.889,149.424
C06694=1156.644,-112.516,-42.550,178.743,5.889,149.424
C06695=1156.649,-112.766,-42.541,178.741,5.889,149.425
C06696=1156.655,-113.016,-42.531,178.739,5.889,149.426
C06697=1156.660,-113.266,-42.522,178.737,5.888,149.426
C06698=1156.666,-113.515,-42.513,178.735,5.888,149.427
C06699=1156.671,-113.765,-42.505,178.733,5.888,149.427
C06700=1156.676,-114.014,-42.496,178.731,5.888,149.428
C06701=1156.682,-114.264,-42.487,178.729,5.887,149.428
C06702=1156.687,-114.514,-42.478,178.727,5.886,149.429
C06703=1156.692,-114.764,-42.469,178.725,5.887,149.429
C06704=1156.698,-115.014,-42.462,178.722,5.886,149.430
C06705=1156.703,-115.264,-42.453,178.721,5.886,149.430
C06706=1156.708,-115.513,-42.444,178.719,5.885,149.431
C06707=1156.714,-115.764,-42.434,178.717,5.885,149.431
C06708=1156.719,-116.014,-42.425,178.714,5.885,149.432
C06709=1156.725,-116.263,-42.417,178.713,5.885,149.433
C06710=1156.730,-116.513,-42.408,178.711,5.884,149.433
C06711=1156.736,-116.762,-42.399,178.709,5.884,149.434
C06712=1156.741,-117.012,-42.390,178.707,5.883,149.434
C06713=1156.747,-117.262,-42.382,178.704,5.883,149.435
C06714=1156.752,-117.512,-42.373,178.702,5.883,149.435
C06715=1156.757,-117.762,-42.365,178.700,5.882,149.436
C06716=1156.762,-118.012,-42.356,178.699,5.882,149.436
C06717=1156.767,-118.261,-42.347,178.696,5.882,149.437
C06718=1156.773,-118.511,-42.338,178.694,5.882,149.437
C06719=1156.778,-118.760,-42.329,178.692,5.881,149.438
C06720=1156.784,-119.011,-42.321,178.691,5.881,149.438
C06721=1156.789,-119.261,-42.312,178.688,5.881,149.439
C06722=1156.795,-119.510,-42.304,178.686,5.881,149.440
C06723=1156.800,-119.760,-42.295,178.684,5.880,149.440
C06724=1156.805,-120.010,-42.286,178.683,5.880,149.441
C06725=1156.811,-120.260,-42.278,178.680,5.879,149.441
C06726=1156.816,-120.509,-42.269,178.679,5.880,149.442
C06727=1156.821,-120.759,-42.260,178.676,5.879,149.442
C06728=1156.827,-121.009,-42.251,178.674,5.879,149.443
C06729=1156.832,-121.259,-42.242,178.672,5.878,149.443
C06730=1156.838,-121.509,-42.235,178.671,5.878,149.444
C06731=1156.843,-121.758,-42.226,178.668,5.878,149.444
C06732=1156.848,-122.008,-42.217,178.667,5.878,149.445
C06733=1156.853,-122.257,-42.209,178.664,5.877,149.445
C06734=1156.859,-122.508,-42.201,178.663,5.877,149.446
C06735=1156.864,-122.757,-42.192,178.660,5.877,149.446
C06736=1156.869,-123.007,-42.183,178.658,5.876,149.447
C06737=1156.875,-123.257,-42.175,178.657,5.876,149.447
C06738=1156.880,-123.507,-42.166,178.654,5.876,149.448
C06739=1156.885,-123.757,-42.157,178.652,5.876,149.449
C06740=1156.891,-124.006,-42.149,178.650,5.875,149.449
C06741=1156.897,-124.256,-42.141,178.649,5.875,149.450
C06742=1156.902,-124.506,-42.132,178.646,5.874,149.450
C06743=1156.908,-124.755,-42.123,178.645,5.874,149.451
C06744=1156.913,-125.006,-42.115,178.642,5.874,149.451
C06745=1156.918,-125.255,-42.107,178.640,5.874,149.452
C06746=1156.923,-125.505,-42.098,178.638,5.873,149.452
C06747=1156.929,-125.755,-42.090,178.637,5.873,149.453
C06748=1156.934,-126.005,-42.081,178.634,5.872,149.453
C06749=1156.939,-126.255,-42.072,178.633,5.872,149.454
C06750=1156.945,-126.504,-42.064,178.630,5.872,149.454
C06751=1156.950,-126.754,-42.055,178.629,5.872,149.455
C06752=1156.955,-127.004,-42.048,178.626,5.871,149.455
C06753=1156.961,-127.254,-42.039,178.625,5.871,149.456
C06754=1156.966,-127.503,-42.030,178.623,5.871,149.456
C06755=1156.972,-127.753,-42.023,178.621,5.871,149.457
C06756=1156.977,-128.003,-42.014,178.618,5.870,149.458
C06757=1156.556,-128.015,-42.056,178.616,5.874,149.459
C06758=1156.551,-127.764,-42.064,178.617,5.874,149.459
C06759=1156.545,-127.515,-42.073,178.619,5.875,149.458
C06760=1156.540,-127.265,-42.081,178.621,5.875,149.458
C06761=1156.535,-127.015,-42.089,178.623,5.875,149.457
C06762=1156.529,-126.766,-42.098,178.625,5.875,149.457
C06763=1156.524,-126.515,-42.106,178.627,5.876,149.456
C06764=1156.518,-126.265,-42.115,178.629,5.876,149.456
C06765=1156.513,-126.016,-42.124,178.631,5.876,149.455
C06766=1156.507,-125.766,-42.132,178.633,5.876,149.455
C06767=1156.502,-125.516,-42.141,178.635,5.877,149.454
C06768=1156.497,-125.267,-42.149,178.637,5.877,149.454
C06769=1156.492,-125.017,-42.157,178.639,5.878,149.453
C06770=1156.486,-124.767,-42.166,178.641,5.877,149.452
C06771=1156.481,-124.518,-42.174,178.643,5.878,149.452
C06772=1156.475,-124.267,-42.182,178.645,5.878,149.451
C06773=1156.470,-124.017,-42.191,178.647,5.879,149.451
C06774=1156.465,-123.767,-42.200,178.648,5.879,149.450
C06775=1156.459,-123.518,-42.208,178.651,5.879,149.450
C06776=1156.454,-123.268,-42.217,178.653,5.879,149.449
C06777=1156.449,-123.018,-42.225,178.655,5.880,149.449
C06778=1156.443,-122.769,-42.233,178.657,5.880,149.448
C06779=1156.438,-122.519,-42.242,178.659,5.881,149.448
C06780=1156.433,-122.269,-42.251,178.660,5.881,149.447
C06781=1156.427,-122.020,-42.259,178.663,5.881,149.447
C06782=1156.422,-121.769,-42.267,178.665,5.881,149.446
C06783=1156.416,-121.519,-42.276,178.667,5.882,149.446
C06784=1156.411,-121.270,-42.285,178.668,5.882,149.445
C06785=1156.405,-121.020,-42.294,178.671,5.882,149.445
C06786=1156.400,-120.770,-42.302,178.673,5.882,149.444
C06787=1156.395,-120.520,-42.311,178.675,5.883,149.443
C06788=1156.390,-120.270,-42.320,178.677,5.884,149.443
C06789=1156.384,-120.021,-42.328,178.679,5.884,149.442
C06790=1156.379,-119.771,-42.337,178.681,5.884,149.442
C06791=1156.373,-119.521,-42.345,178.682,5.884,149.441
C06792=1156.368,-119.271,-42.354,178.685,5.885,149.441
C06793=1156.362,-119.022,-42.363,178.687,5.885,149.440
C06794=1156.357,-118.772,-42.372,178.689,5.885,149.440
C06795=1156.352,-118.522,-42.381,178.691,5.885,149.439
C06796=1156.347,-118.272,-42.390,178.693,5.886,149.439
C06797=1156.341,-118.022,-42.397,178.695,5.886,149.438
C06798=1156.336,-117.773,-42.406,178.697,5.886,149.438
C06799=1156.330,-117.523,-42.415,178.699,5.886,149.437
C06800=1156.325,-117.273,-42.424,178.701,5.887,149.437
C06801=1156.319,-117.024,-42.433,178.703,5.887,149.436
C06802=1156.314,-116.774,-42.441,178.705,5.887,149.435
C06803=1156.309,-116.523,-42.450,178.707,5.887,149.435
C06804=1156.304,-116.274,-42.459,178.709,5.888,149.434
C06805=1156.298,-116.024,-42.467,178.711,5.889,149.434
C06806=1156.293,-115.775,-42.476,178.713,5.888,149.433
C06807=1156.288,-115.525,-42.485,178.715,5.889,149.433
C06808=1156.282,-115.275,-42.494,178.717,5.889,149.432
C06809=1156.277,-115.025,-42.503,178.719,5.890,149.432
C06810=1156.272,-114.775,-42.512,178.721,5.890,149.431
C06811=1156.266,-114.526,-42.520,178.723,5.890,149.431
C06812=1156.260,-114.276,-42.530,178.725,5.890,149.430
C06813=1156.255,-114.026,-42.538,178.727,5.891,149.430
C06814=1156.250,-113.776,-42.547,178.729,5.891,149.429
C06815=1156.245,-113.526,-42.556,178.731,5.891,149.428
C06816=1156.239,-113.277,-42.564,178.734,5.892,149.428
C06817=1156.234,-113.027,-42.573,178.735,5.892,149.427
C06818=1156.228,-112.777,-42.582,178.737,5.893,149.427
C06819=1156.223,-112.527,-42.591,178.739,5.893,149.426
C06820=1156.218,-112.277,-42.600,178.742,5.893,149.426
C06821=1156.212,-112.027,-42.609,178.743,5.893,149.425
C06822=1156.206,-111.778,-42.618,178.746,5.894,149.425
C06823=1156.201,-111.528,-42.627,178.747,5.894,149.424
C06824=1156.196,-111.278,-42.636,178.750,5.894,149.424
C06825=1156.191,-111.028,-42.644,178.752,5.895,149.423
C06826=1156.186,-110.778,-42.653,178.754,5.895,149.423
C06827=1156.181,-110.529,-42.662,178.756,5.896,149.422
C06828=1156.175,-110.278,-42.672,178.758,5.895,149.421
C06829=1156.169,-110.029,-42.680,178.760,5.896,149.421
C06830=1156.164,-109.780,-42.690,178.762,5.896,149.420
C06831=1156.159,-109.530,-42.699,178.764,5.897,149.420
C06832=1156.154,-109.280,-42.708,178.766,5.896,149.419
C06833=1156.149,-109.030,-42.717,178.768,5.897,149.419
C06834=1156.143,-108.780,-42.726,178.770,5.898,149.418
C06835=1156.138,-108.530,-42.735,178.772,5.898,149.418
C06836=1156.132,-108.281,-42.744,178.775,5.898,149.417
C06837=1156.127,-108.031,-42.752,178.776,5.898,149.417
C06838=1156.121,-107.782,-42.761,178.778,5.899,149.416
C06839=1156.116,-107.531,-42.771,178.780,5.899,149.416
C06840=1156.110,-107.282,-42.780,178.783,5.899,149.415
C06841=1156.105,-107.032,-42.789,178.785,5.900,149.414
C06842=1156.100,-106.782,-42.798,178.786,5.900,149.414
C06843=1156.095,-106.533,-42.807,178.789,5.901,149.413
C06844=1156.089,-106.282,-42.817,178.791,5.900,149.413
C06845=1156.084,-106.033,-42.825,178.793,5.901,149.412
C06846=1156.079,-105.783,-42.834,178.795,5.901,149.412
C06847=1156.074,-105.533,-42.843,178.797,5.902,149.411
C06848=1156.067,-105.283,-42.852,178.799,5.902,149.411
C06849=1156.062,-105.034,-42.862,178.801,5.902,149.410
C06850=1156.057,-104.784,-42.871,178.803,5.903,149.410
C06851=1156.052,-104.535,-42.880,178.805,5.903,149.409
C06852=1156.046,-104.284,-42.889,178.807,5.903,149.408
C06853=1156.041,-104.034,-42.898,178.810,5.904,149.408
C06854=1156.036,-103.785,-42.908,178.811,5.904,149.407
C06855=1156.031,-103.535,-42.917,178.814,5.904,149.407
C06856=1156.025,-103.285,-42.926,178.816,5.904,149.406
C06857=1156.020,-103.035,-42.935,178.818,5.905,149.406
C06858=1156.014,-102.763,-42.945,178.820,5.905,149.405
C06859=1156.009,-102.492,-42.956,178.822,5.905,149.405
C06860=1156.003,-102.220,-42.965,178.825,5.906,149.404
C06861=1155.996,-101.947,-42.976,178.827,5.907,149.403
C06862=1155.991,-101.698,-42.984,178.828,5.906,149.403
C06863=1155.986,-101.448,-42.994,178.831,5.907,149.402
C06864=1155.980,-101.198,-43.004,178.833,5.908,149.402
C06865=1155.975,-100.948,-43.012,178.835,5.908,149.401
C06866=1155.970,-100.699,-43.022,178.837,5.908,149.401
C06867=1155.965,-100.449,-43.031,178.839,5.908,149.400
C06868=1155.959,-100.199,-43.040,178.841,5.909,149.399
C06869=1155.954,-99.949,-43.049,178.844,5.909,149.399
C06870=1155.948,-99.700,-43.060,178.846,5.909,149.398
C06871=1155.943,-99.450,-43.068,178.848,5.910,149.398
C06872=1155.938,-99.200,-43.077,178.850,5.911,149.397
C06873=1155.933,-98.950,-43.088,178.852,5.910,149.397
C06874=1155.927,-98.701,-43.096,178.854,5.911,149.396
C06875=1155.922,-98.451,-43.105,178.856,5.911,149.396
C06876=1155.917,-98.201,-43.116,178.858,5.912,149.395
C06877=1155.911,-97.951,-43.124,178.861,5.912,149.394
C06878=1155.906,-97.701,-43.134,178.862,5.912,149.394
C06879=1155.901,-97.452,-43.144,178.865,5.913,149.393
C06880=1155.896,-97.202,-43.152,178.867,5.912,149.393
C06881=1155.890,-96.953,-43.163,178.869,5.913,149.392
C06882=1155.885,-96.703,-43.172,178.871,5.914,149.392
C06883=1155.879,-96.453,-43.181,178.873,5.913,149.391
C06884=1155.874,-96.203,-43.191,178.875,5.914,149.391
C06885=1155.869,-95.952,-43.201,178.878,5.915,149.390
C06886=1155.864,-95.703,-43.210,178.879,5.915,149.390
C06887=1155.859,-95.453,-43.219,178.882,5.915,149.389
C06888=1155.853,-95.203,-43.229,178.883,5.915,149.388
C06889=1155.848,-94.954,-43.238,178.886,5.916,149.388
C06890=1155.842,-94.704,-43.248,178.888,5.916,149.387
C06891=1155.837,-94.455,-43.257,178.890,5.916,149.387
C06892=1155.831,-94.204,-43.267,178.892,5.917,149.386
C06893=1155.826,-93.955,-43.276,178.895,5.918,149.386
C06894=1155.820,-93.705,-43.286,178.896,5.918,149.385
C06895=1155.816,-93.456,-43.295,178.898,5.918,149.385
C06896=1155.810,-93.206,-43.305,178.901,5.918,149.384
C06897=1155.805,-92.956,-43.315,178.903,5.919,149.383
C06898=1155.799,-92.706,-43.324,178.905,5.919,149.383
C06899=1155.795,-92.456,-43.334,178.907,5.919,149.382
C06900=1155.789,-92.206,-43.344,178.909,5.920,149.382
C06901=1155.784,-91.957,-43.353,178.911,5.921,149.381
C06902=1155.778,-91.707,-43.363,178.913,5.920,149.380
C06903=1155.773,-91.458,-43.372,178.916,5.921,149.380
C06904=1155.767,-91.207,-43.382,178.918,5.922,149.380
C06905=1155.762,-90.958,-43.391,178.920,5.921,149.379
C06906=1155.756,-90.708,-43.401,178.922,5.922,149.378
C06907=1155.752,-90.459,-43.410,178.924,5.922,149.378
C06908=1155.746,-90.208,-43.420,178.926,5.922,149.377
C06909=1155.741,-89.959,-43.430,178.929,5.923,149.377
C06910=1155.736,-89.709,-43.440,178.930,5.923,149.376
C06911=1155.731,-89.459,-43.449,178.933,5.923,149.375
C06912=1155.725,-89.210,-43.459,178.935,5.924,149.375
C06913=1155.720,-88.960,-43.468,178.937,5.924,149.374
C06914=1155.714,-88.710,-43.478,178.939,5.925,149.374
C06915=1155.709,-88.461,-43.489,178.942,5.925,149.373
C06916=1155.704,-88.210,-43.498,178.943,5.925,149.373
C06917=1155.699,-87.961,-43.508,178.946,5.926,149.372
C06918=1155.694,-87.711,-43.518,178.948,5.926,149.372
C06919=1155.688,-87.461,-43.527,178.950,5.926,149.371
C06920=1155.682,-87.212,-43.537,178.952,5.927,149.370
C06921=1155.677,-86.962,-43.546,178.954,5.928,149.370
C06922=1155.672,-86.712,-43.557,178.956,5.928,149.369
C06923=1155.667,-86.462,-43.566,178.959,5.928,149.369
C06924=1155.661,-86.212,-43.576,178.961,5.929,149.368
C06925=1155.656,-85.963,-43.586,178.963,5.929,149.368
C06926=1155.651,-85.713,-43.596,178.965,5.929,149.367
C06927=1155.646,-85.463,-43.606,178.967,5.930,149.367
C06928=1155.641,-85.213,-43.615,178.969,5.930,149.366
C06929=1155.635,-84.964,-43.625,178.972,5.930,149.365
C06930=1155.629,-84.714,-43.636,178.974,5.931,149.365
C06931=1155.624,-84.464,-43.645,178.975,5.931,149.364
C06932=1155.619,-84.214,-43.655,178.978,5.931,149.364
C06933=1155.614,-83.965,-43.665,178.980,5.932,149.363
C06934=1155.609,-83.715,-43.675,178.982,5.932,149.363
C06935=1155.603,-83.465,-43.684,178.985,5.932,149.362
C06936=1155.597,-83.216,-43.695,178.987,5.933,149.362
C06937=1155.593,-82.966,-43.705,178.989,5.933,149.361
C06938=1155.587,-82.716,-43.715,178.991,5.934,149.360
C06939=1155.582,-82.466,-43.724,178.993,5.934,149.360
C06940=1155.577,-82.217,-43.734,178.995,5.934,149.359
C06941=1155.572,-81.967,-43.744,178.997,5.935,149.359
C06942=1155.566,-81.717,-43.755,179.000,5.936,149.358
C06943=1155.560,-81.468,-43.765,179.002,5.935,149.357
C06944=1155.555,-81.218,-43.774,179.004,5.936,149.357
C06945=1155.550,-80.967,-43.784,179.006,5.937,149.357
C06946=1155.545,-80.718,-43.795,179.009,5.937,149.356
C06947=1155.540,-80.469,-43.804,179.010,5.937,149.355
C06948=1155.534,-80.219,-43.814,179.013,5.937,149.355
C06949=1155.529,-79.969,-43.825,179.015,5.938,149.354
C06950=1155.523,-79.719,-43.834,179.017,5.938,149.354
C06951=1155.519,-79.469,-43.844,179.020,5.939,149.353
C06952=1155.513,-79.220,-43.854,179.022,5.939,149.352
C06953=1155.508,-78.970,-43.865,179.023,5.939,149.352
C06954=1155.502,-78.720,-43.875,179.026,5.940,149.351
C06955=1155.497,-78.471,-43.885,179.028,5.940,149.351
C06956=1155.492,-78.221,-43.895,179.031,5.941,149.350
C06957=1155.487,-77.971,-43.905,179.032,5.941,149.350
C06958=1155.481,-77.722,-43.916,179.035,5.942,149.349
C06959=1155.475,-77.471,-43.925,179.037,5.942,149.348
C06960=1155.470,-77.221,-43.936,179.039,5.942,149.348
C06961=1155.466,-76.972,-43.945,179.041,5.943,149.347
C06962=1155.460,-76.700,-43.957,179.044,5.943,149.347
C06963=1155.454,-76.430,-43.967,179.046,5.943,149.346
C06964=1155.448,-76.158,-43.979,179.049,5.944,149.346
C06965=1155.443,-75.887,-43.990,179.051,5.944,149.345
C06966=1155.437,-75.637,-44.000,179.053,5.945,149.344
C06967=1155.431,-75.388,-44.010,179.056,5.945,149.344
C06968=1155.426,-75.138,-44.021,179.058,5.946,149.343
C06969=1155.421,-74.888,-44.031,179.059,5.946,149.343
C06970=1155.415,-74.638,-44.041,179.062,5.946,149.342
C06971=1155.411,-74.388,-44.051,179.064,5.947,149.341
C06972=1155.405,-74.139,-44.062,179.066,5.948,149.341
C06973=1155.400,-73.889,-44.072,179.068,5.947,149.340
C06974=1155.395,-73.639,-44.082,179.071,5.948,149.340
C06975=1155.389,-73.390,-44.093,179.073,5.948,149.339
C06976=1155.384,-73.140,-44.103,179.075,5.948,149.339
C06977=1155.379,-72.890,-44.113,179.077,5.949,149.338
C06978=1155.373,-72.640,-44.124,179.080,5.950,149.337
C06979=1155.367,-72.391,-44.134,179.082,5.950,149.337
C06980=1155.363,-72.141,-44.144,179.084,5.950,149.336
C06981=1155.358,-71.891,-44.154,179.086,5.951,149.336
C06982=1155.353,-71.641,-44.165,179.088,5.952,149.335
C06983=1155.347,-71.391,-44.175,179.091,5.952,149.335
C06984=1155.342,-71.143,-44.186,179.093,5.952,149.334
C06985=1155.337,-70.892,-44.196,179.095,5.952,149.333
C06986=1155.331,-70.643,-44.206,179.098,5.953,149.333
C06987=1155.326,-70.393,-44.217,179.100,5.954,149.332
C06988=1155.321,-70.143,-44.227,179.102,5.953,149.332
C06989=1155.315,-69.893,-44.237,179.104,5.954,149.331
C06990=1155.310,-69.643,-44.248,179.107,5.955,149.331
C06991=1155.304,-69.394,-44.258,179.108,5.955,149.330
C06992=1155.299,-69.145,-44.269,179.110,5.955,149.330
C06993=1155.294,-68.894,-44.280,179.113,5.956,149.329
C06994=1155.288,-68.645,-44.290,179.115,5.957,149.328
C06995=1155.283,-68.395,-44.300,179.117,5.956,149.328
C06996=1155.278,-68.145,-44.311,179.120,5.957,149.327
C06997=1155.273,-67.895,-44.321,179.122,5.958,149.327
C06998=1155.268,-67.646,-44.332,179.124,5.958,149.326
C06999=1155.262,-67.396,-44.342,179.126,5.958,149.326
C07000=1155.257,-67.146,-44.353,179.129,5.958,149.325
C07001=1155.251,-66.897,-44.363,179.131,5.959,149.324
C07002=1155.246,-66.646,-44.374,179.133,5.960,149.324
C07003=1155.241,-66.397,-44.385,179.136,5.960,149.323
C07004=1155.236,-66.147,-44.395,179.137,5.960,149.323
C07005=1155.230,-65.898,-44.405,179.140,5.961,149.322
C07006=1155.225,-65.647,-44.416,179.142,5.962,149.321
C07007=1155.220,-65.399,-44.427,179.145,5.962,149.321
C07008=1155.215,-65.149,-44.437,179.146,5.962,149.320
C07009=1155.210,-64.899,-44.448,179.149,5.963,149.320
C07010=1155.204,-64.650,-44.459,179.151,5.963,149.319
C07011=1155.199,-64.400,-44.469,179.154,5.964,149.319
C07012=1155.194,-64.150,-44.479,179.156,5.964,149.318
C07013=1155.189,-63.900,-44.490,179.158,5.964,149.317
C07014=1155.183,-63.651,-44.501,179.160,5.965,149.317
C07015=1155.178,-63.401,-44.512,179.163,5.965,149.316
C07016=1155.173,-63.151,-44.522,179.165,5.966,149.316
C07017=1155.167,-62.901,-44.534,179.167,5.966,149.315
C07018=1155.162,-62.652,-44.544,179.169,5.967,149.315
C07019=1155.157,-62.401,-44.554,179.172,5.967,149.314
C07020=1155.151,-62.152,-44.565,179.174,5.968,149.313
C07021=1155.146,-61.902,-44.576,179.176,5.968,149.313
C07022=1155.141,-61.653,-44.587,179.178,5.968,149.312
C07023=1155.136,-61.403,-44.597,179.180,5.969,149.312
C07024=1155.131,-61.153,-44.608,179.183,5.969,149.311
C07025=1155.126,-60.904,-44.619,179.185,5.970,149.311
C07026=1155.120,-60.653,-44.630,179.187,5.970,149.310
C07027=1155.115,-60.404,-44.641,179.190,5.971,149.309
C07028=1155.110,-60.154,-44.652,179.192,5.971,149.309
C07029=1155.104,-59.905,-44.662,179.194,5.972,149.308
C07030=1155.100,-59.655,-44.673,179.197,5.973,149.308
C07031=1155.094,-59.405,-44.683,179.199,5.972,149.307
C07032=1155.089,-59.156,-44.695,179.201,5.973,149.307
C07033=1155.083,-58.906,-44.705,179.204,5.973,149.306
C07034=1155.078,-58.656,-44.717,179.206,5.974,149.305
C07035=1155.073,-58.406,-44.727,179.207,5.974,149.305
C07036=1155.068,-58.157,-44.738,179.210,5.974,149.304
C07037=1155.063,-57.907,-44.749,179.212,5.975,149.304
C07038=1155.057,-57.657,-44.760,179.215,5.976,149.303
C07039=1155.052,-57.407,-44.771,179.217,5.976,149.303
C07040=1155.046,-57.158,-44.781,179.220,5.977,149.302
C07041=1155.042,-56.908,-44.792,179.221,5.977,149.301
C07042=1155.037,-56.659,-44.804,179.224,5.977,149.301
C07043=1155.031,-56.409,-44.814,179.226,5.978,149.300
C07044=1155.026,-56.159,-44.826,179.228,5.979,149.300
C07045=1155.020,-55.910,-44.836,179.231,5.979,149.299
C07046=1155.016,-55.660,-44.847,179.233,5.979,149.298
C07047=1155.011,-55.410,-44.858,179.235,5.980,149.298
C07048=1155.005,-55.160,-44.869,179.237,5.980,149.297
C07049=1155.000,-54.910,-44.880,179.240,5.981,149.297
C07050=1154.995,-54.661,-44.891,179.242,5.982,149.296
C07051=1154.990,-54.412,-44.902,179.244,5.982,149.296
C07052=1154.984,-54.161,-44.913,179.247,5.982,149.295
C07053=1154.979,-53.912,-44.924,179.249,5.983,149.294
C07054=1154.974,-53.662,-44.935,179.251,5.983,149.294
C07055=1154.968,-53.412,-44.947,179.254,5.984,149.293
C07056=1154.963,-53.163,-44.958,179.256,5.984,149.293
C07057=1154.958,-52.913,-44.968,179.258,5.984,149.292
C07058=1154.952,-52.663,-44.980,179.260,5.985,149.291
C07059=1154.947,-52.414,-44.991,179.263,5.986,149.291
C07060=1154.942,-52.164,-45.002,179.265,5.986,149.290
C07061=1154.937,-51.914,-45.013,179.268,5.987,149.290
C07062=1154.931,-51.664,-45.024,179.270,5.988,149.289
C07063=1154.926,-51.415,-45.035,179.272,5.987,149.289
C07064=1154.922,-51.165,-45.046,179.274,5.988,149.288
C07065=1154.916,-50.916,-45.058,179.277,5.988,149.287
C07066=1154.910,-50.645,-45.070,179.279,5.989,149.287
C07067=1154.905,-50.374,-45.082,179.282,5.990,149.286
C07068=1154.899,-50.104,-45.094,179.284,5.990,149.285
C07069=1154.893,-49.833,-45.106,179.286,5.991,149.285
C07070=1154.887,-49.584,-45.117,179.289,5.991,149.284
C07071=1154.883,-49.334,-45.129,179.291,5.992,149.284
C07072=1154.878,-49.084,-45.139,179.294,5.992,149.283
C07073=1154.872,-48.834,-45.151,179.295,5.992,149.283
C07074=1154.867,-48.585,-45.162,179.298,5.993,149.282
C07075=1154.862,-48.335,-45.174,179.300,5.993,149.281
C07076=1154.857,-48.085,-45.184,179.303,5.994,149.281
C07077=1154.851,-47.836,-45.195,179.305,5.995,149.280
C07078=1154.846,-47.586,-45.207,179.307,5.995,149.280
C07079=1154.841,-47.336,-45.219,179.310,5.996,149.279
C07080=1154.835,-47.086,-45.230,179.312,5.996,149.279
C07081=1154.830,-46.837,-45.241,179.314,5.996,149.278
C07082=1154.825,-46.587,-45.252,179.316,5.997,149.277
C07083=1154.820,-46.337,-45.264,179.319,5.997,149.277
C07084=1154.815,-46.088,-45.275,179.321,5.998,149.276
C07085=1154.809,-45.838,-45.287,179.324,5.999,149.276
C07086=1154.804,-45.588,-45.297,179.326,5.999,149.275
C07087=1154.799,-45.338,-45.309,179.328,5.999,149.274
C07088=1154.794,-45.089,-45.320,179.330,6.000,149.274
C07089=1154.788,-44.839,-45.332,179.333,6.000,149.273
C07090=1154.783,-44.590,-45.343,179.335,6.001,149.273
C07091=1154.778,-44.340,-45.355,179.337,6.002,149.272
C07092=1154.773,-44.090,-45.366,179.340,6.002,149.272
C07093=1154.767,-43.841,-45.378,179.342,6.003,149.271
C07094=1154.763,-43.591,-45.389,179.345,6.003,149.270
C07095=1154.757,-43.341,-45.400,179.347,6.003,149.270
C07096=1154.752,-43.091,-45.412,179.349,6.004,149.269
C07097=1154.746,-42.842,-45.423,179.351,6.005,149.269
C07098=1154.741,-42.592,-45.434,179.354,6.005,149.268
C07099=1154.736,-42.342,-45.446,179.356,6.006,149.268
C07100=1154.731,-42.093,-45.458,179.359,6.006,149.267
C07101=1154.726,-41.843,-45.469,179.361,6.007,149.266
C07102=1154.720,-41.593,-45.481,179.364,6.007,149.266
C07103=1154.715,-41.344,-45.492,179.366,6.008,149.265
C07104=1154.710,-41.094,-45.504,179.368,6.008,149.265
C07105=1154.705,-40.844,-45.515,179.370,6.009,149.264
C07106=1154.700,-40.594,-45.527,179.372,6.009,149.264
C07107=1154.695,-40.345,-45.539,179.375,6.010,149.263
C07108=1154.689,-40.095,-45.550,179.377,6.011,149.262
C07109=1154.683,-39.846,-45.562,179.380,6.011,149.262
C07110=1154.679,-39.596,-45.573,179.382,6.012,149.261
C07111=1154.673,-39.346,-45.585,179.385,6.012,149.260
C07112=1154.669,-39.096,-45.596,179.387,6.013,149.260
C07113=1154.663,-38.846,-45.608,179.390,6.013,149.259
C07114=1154.657,-38.597,-45.620,179.391,6.013,149.259
C07115=1154.652,-38.348,-45.631,179.394,6.014,149.258
C07116=1154.647,-38.098,-45.644,179.396,6.015,149.258
C07117=1154.642,-37.848,-45.656,179.399,6.015,149.257
C07118=1154.637,-37.599,-45.667,179.401,6.016,149.257
C07119=1154.632,-37.349,-45.679,179.404,6.016,149.256
C07120=1154.627,-37.099,-45.690,179.406,6.017,149.255
C07121=1154.621,-36.850,-45.702,179.408,6.018,149.255
C07122=1154.616,-36.600,-45.714,179.411,6.018,149.254
C07123=1154.611,-36.350,-45.725,179.413,6.019,149.254
C07124=1154.606,-36.100,-45.737,179.415,6.020,149.253
C07125=1154.600,-35.851,-45.749,179.417,6.020,149.253
C07126=1154.596,-35.601,-45.761,179.420,6.020,149.252
C07127=1154.590,-35.352,-45.772,179.422,6.021,149.251
C07128=1154.585,-35.102,-45.784,179.425,6.021,149.251
C07129=1154.579,-34.852,-45.796,179.427,6.022,149.250
C07130=1154.575,-34.602,-45.808,179.429,6.022,149.249
C07131=1154.569,-34.353,-45.820,179.432,6.023,149.249
C07132=1154.564,-34.103,-45.832,179.434,6.024,149.248
C07133=1154.559,-33.854,-45.843,179.436,6.024,149.248
C07134=1154.553,-33.604,-45.855,179.439,6.025,149.247
C07135=1154.548,-33.354,-45.867,179.441,6.026,149.247
C07136=1154.543,-33.105,-45.879,179.444,6.026,149.246
C07137=1154.538,-32.855,-45.891,179.446,6.027,149.245
C07138=1154.533,-32.605,-45.903,179.449,6.027,149.245
C07139=1154.527,-32.355,-45.914,179.451,6.028,149.244
C07140=1154.522,-32.106,-45.927,179.453,6.028,149.244
C07141=1154.518,-31.856,-45.938,179.455,6.028,149.243
C07142=1154.512,-31.606,-45.950,179.458,6.029,149.242
C07143=1154.507,-31.357,-45.963,179.460,6.030,149.242
C07144=1154.502,-31.107,-45.975,179.463,6.030,149.241
C07145=1154.496,-30.857,-45.987,179.465,6.031,149.241
C07146=1154.492,-30.608,-45.999,179.468,6.031,149.240
C07147=1154.486,-30.358,-46.010,179.470,6.032,149.240
C07148=1154.481,-30.108,-46.022,179.472,6.033,149.239
C07149=1154.476,-29.859,-46.035,179.475,6.033,149.238
C07150=1154.470,-29.609,-46.047,179.477,6.034,149.238
C07151=1154.466,-29.359,-46.058,179.479,6.035,149.237
C07152=1154.461,-29.110,-46.071,179.482,6.035,149.237
C07153=1154.455,-28.860,-46.083,179.484,6.036,149.236
C07154=1154.450,-28.610,-46.094,179.486,6.037,149.236
C07155=1154.445,-28.361,-46.107,179.489,6.037,149.235
C07156=1154.439,-28.111,-46.119,179.491,6.038,149.234
C07157=1154.435,-27.862,-46.131,179.494,6.038,149.234
C07158=1154.429,-27.612,-46.143,179.496,6.039,149.233
C07159=1154.424,-27.362,-46.155,179.499,6.039,149.233
C07160=1154.419,-27.113,-46.167,179.501,6.040,149.232
C07161=1154.413,-26.863,-46.179,179.504,6.041,149.231
C07162=1154.408,-26.613,-46.192,179.505,6.041,149.231
C07163=1154.403,-26.363,-46.204,179.508,6.041,149.230
C07164=1154.398,-26.114,-46.216,179.510,6.042,149.230
C07165=1154.393,-25.865,-46.228,179.513,6.042,149.229
C07166=1154.388,-25.615,-46.239,179.515,6.043,149.229
C07167=1154.382,-25.365,-46.252,179.518,6.044,149.228
C07168=1154.377,-25.115,-46.264,179.520,6.044,149.227
C07169=1154.372,-24.866,-46.277,179.522,6.045,149.227
C07170=1154.367,-24.596,-46.290,179.525,6.046,149.226
C07171=1154.360,-24.326,-46.303,179.528,6.047,149.226
C07172=1154.355,-24.056,-46.316,179.531,6.047,149.225
C07173=1154.350,-23.786,-46.329,179.533,6.048,149.224
C07174=1154.344,-23.536,-46.342,179.535,6.048,149.224
C07175=1154.339,-23.286,-46.354,179.538,6.049,149.223
C07176=1154.334,-23.037,-46.366,179.540,6.050,149.223
C07177=1154.329,-22.788,-46.379,179.542,6.050,149.222
C07178=1154.323,-22.538,-46.391,179.545,6.051,149.221
C07179=1154.318,-22.288,-46.404,179.547,6.052,149.221
C07180=1154.313,-22.039,-46.415,179.550,6.052,149.220
C07181=1154.308,-21.789,-46.428,179.552,6.053,149.220
C07182=1154.303,-21.540,-46.441,179.555,6.053,149.219
C07183=1154.298,-21.289,-46.453,179.557,6.054,149.219
C07184=1154.293,-21.040,-46.465,179.560,6.055,149.218
C07185=1154.287,-20.790,-46.477,179.562,6.055,149.217
C07186=1154.282,-20.541,-46.490,179.564,6.056,149.217
C07187=1154.277,-20.291,-46.503,179.567,6.057,149.216
C07188=1154.271,-20.041,-46.514,179.569,6.057,149.216
C07189=1154.266,-19.792,-46.527,179.571,6.058,149.215
C07190=1154.261,-19.543,-46.540,179.574,6.058,149.214
C07191=1154.256,-19.292,-46.552,179.576,6.059,149.214
C07192=1154.251,-19.043,-46.565,179.579,6.059,149.213
C07193=1154.246,-18.794,-46.577,179.581,6.060,149.213
C07194=1154.241,-18.544,-46.589,179.584,6.061,149.212
C07195=1154.235,-18.294,-46.602,179.586,6.062,149.212
C07196=1154.230,-18.045,-46.615,179.589,6.062,149.211
C07197=1154.225,-17.795,-46.628,179.591,6.063,149.210
C07198=1154.220,-17.545,-46.640,179.593,6.063,149.210
C07199=1154.215,-17.295,-46.652,179.596,6.064,149.209
C07200=1154.210,-17.046,-46.665,179.598,6.064,149.209
C07201=1154.204,-16.797,-46.677,179.601,6.065,149.208
C07202=1154.199,-16.547,-46.689,179.603,6.066,149.207
C07203=1154.194,-16.297,-46.702,179.605,6.066,149.207
C07204=1154.189,-16.047,-46.715,179.608,6.067,149.206
C07205=1154.183,-15.798,-46.728,179.610,6.068,149.206
C07206=1154.178,-15.548,-46.740,179.613,6.068,149.205
C07207=1154.173,-15.299,-46.753,179.615,6.069,149.205
C07208=1154.168,-15.049,-46.766,179.618,6.069,149.204
C07209=1154.163,-14.799,-46.778,179.620,6.070,149.203
C07210=1154.158,-14.550,-46.791,179.623,6.071,149.203
C07211=1154.152,-14.300,-46.804,179.625,6.071,149.202
C07212=1154.147,-14.050,-46.816,179.628,6.073,149.202
C07213=1154.142,-13.800,-46.829,179.630,6.073,149.201
C07214=1154.137,-13.551,-46.841,179.633,6.074,149.200
C07215=1154.132,-13.302,-46.854,179.635,6.075,149.200
C07216=1154.127,-13.052,-46.867,179.638,6.075,149.199
C07217=1154.122,-12.802,-46.880,179.640,6.076,149.199
C07218=1154.117,-12.553,-46.893,179.642,6.076,149.198
C07219=1154.111,-12.303,-46.905,179.645,6.077,149.198
C07220=1154.107,-12.053,-46.918,179.647,6.078,149.197
C07221=1154.101,-11.803,-46.930,179.649,6.078,149.196
C07222=1154.096,-11.554,-46.943,179.652,6.079,149.196
C07223=1154.091,-11.305,-46.956,179.654,6.080,149.195
C07224=1154.086,-11.055,-46.969,179.657,6.080,149.195
C07225=1154.081,-10.805,-46.982,179.659,6.081,149.194
C07226=1154.075,-10.556,-46.995,179.662,6.081,149.193
C07227=1154.070,-10.306,-47.007,179.664,6.082,149.193
C07228=1154.065,-10.056,-47.020,179.667,6.083,149.192
C07229=1154.060,-9.807,-47.033,179.669,6.083,149.192
C07230=1154.054,-9.557,-47.046,179.672,6.085,149.191
C07231=1154.050,-9.307,-47.059,179.674,6.085,149.191
C07232=1154.045,-9.058,-47.072,179.677,6.086,149.190
C07233=1154.039,-8.808,-47.085,179.679,6.087,149.190
C07234=1154.034,-8.558,-47.098,179.682,6.087,149.189
C07235=1154.029,-8.309,-47.110,179.684,6.088,149.188
C07236=1154.024,-8.060,-47.123,179.687,6.088,149.188
C07237=1154.019,-7.809,-47.137,179.689,6.089,149.187
C07238=1154.014,-7.560,-47.149,179.691,6.090,149.187
C07239=1154.009,-7.311,-47.162,179.694,6.090,149.186
C07240=1154.004,-7.061,-47.176,179.696,6.091,149.185
C07241=1153.999,-6.812,-47.189,179.698,6.092,149.185
C07242=1153.993,-6.562,-47.201,179.701,6.092,149.184
C07243=1153.988,-6.312,-47.215,179.704,6.094,149.184
C07244=1153.983,-6.063,-47.227,179.707,6.094,149.183
C07245=1153.977,-5.813,-47.241,179.709,6.095,149.183
C07246=1153.973,-5.563,-47.254,179.711,6.095,149.182
C07247=1153.967,-5.314,-47.266,179.714,6.096,149.181
C07248=1153.962,-5.065,-47.280,179.716,6.097,149.181
C07249=1153.957,-4.815,-47.293,179.718,6.097,149.180
C07250=1153.952,-4.565,-47.306,179.721,6.098,149.180
C07251=1153.947,-4.315,-47.319,179.723,6.099,149.179
C07252=1153.942,-4.066,-47.332,179.726,6.099,149.178
C07253=1153.936,-3.816,-47.345,179.729,6.101,149.178
C07254=1153.932,-3.567,-47.359,179.731,6.101,149.177
C07255=1153.926,-3.317,-47.372,179.733,6.102,149.177
C07256=1153.921,-3.067,-47.385,179.736,6.102,149.176
C07257=1153.916,-2.818,-47.398,179.738,6.103,149.176
C07258=1153.910,-2.568,-47.411,179.741,6.104,149.175
C07259=1153.906,-2.319,-47.424,179.743,6.105,149.174
C07260=1153.900,-2.069,-47.438,179.745,6.105,149.174
C07261=1153.896,-1.819,-47.451,179.748,6.106,149.173
C07262=1153.890,-1.569,-47.464,179.751,6.107,149.173
C07263=1153.885,-1.321,-47.477,179.753,6.108,149.172
C07264=1153.880,-1.070,-47.491,179.756,6.109,149.172
C07265=1153.875,-0.821,-47.503,179.758,6.109,149.171
C07266=1153.870,-0.571,-47.518,179.760,6.110,149.171
C07267=1153.865,-0.322,-47.530,179.763,6.110,149.170
C07268=1153.859,-0.072,-47.544,179.765,6.111,149.169
C07269=1153.855,0.177,-47.557,179.768,6.112,149.169
C07270=1153.849,0.427,-47.571,179.771,6.113,149.168
C07271=1153.844,0.677,-47.583,179.773,6.114,149.168
C07272=1153.839,0.926,-47.597,179.775,6.115,149.167
C07273=1153.834,1.176,-47.610,179.778,6.115,149.166
C07274=1153.828,1.446,-47.624,179.781,6.115,149.166
C07275=1153.822,1.714,-47.639,179.784,6.117,149.165
C07276=1153.818,1.983,-47.653,179.786,6.117,149.165
C07277=1153.812,2.254,-47.668,179.789,6.118,149.164
C07278=1153.806,2.503,-47.682,179.791,6.119,149.163
C07279=1153.802,2.753,-47.694,179.794,6.119,149.163
C07280=1153.796,3.002,-47.708,179.796,6.121,149.162
C07281=1153.791,3.252,-47.722,179.799,6.121,149.162
C07282=1153.786,3.501,-47.735,179.801,6.122,149.161
C07283=1153.781,3.751,-47.749,179.804,6.122,149.160
C07284=1153.776,4.000,-47.761,179.806,6.123,149.160
C07285=1153.771,4.250,-47.776,179.809,6.124,149.159
C07286=1153.765,4.500,-47.789,179.812,6.125,149.159
C07287=1153.761,4.749,-47.803,179.814,6.126,149.158
C07288=1153.755,4.999,-47.816,179.816,6.127,149.158
C07289=1153.751,5.248,-47.829,179.819,6.127,149.157
C07290=1153.745,5.498,-47.843,179.821,6.128,149.157
C07291=1153.740,5.747,-47.857,179.824,6.128,149.156
C07292=1153.735,5.997,-47.870,179.826,6.129,149.155
C07293=1153.730,6.246,-47.884,179.829,6.130,149.155
C07294=1153.725,6.497,-47.897,179.831,6.131,149.154
C07295=1153.720,6.745,-47.911,179.834,6.132,149.154
C07296=1153.715,6.996,-47.924,179.836,6.133,149.153
C07297=1153.709,7.245,-47.938,179.839,6.133,149.152
C07298=1153.705,7.494,-47.952,179.841,6.134,149.152
C07299=1153.699,7.744,-47.965,179.844,6.135,149.151
C07300=1153.694,7.993,-47.979,179.846,6.136,149.151
C07301=1153.689,8.243,-47.992,179.849,6.137,149.150
C07302=1153.684,8.492,-48.006,179.851,6.137,149.150
C07303=1153.679,8.742,-48.020,179.853,6.138,149.149
C07304=1153.673,8.992,-48.034,179.857,6.139,149.149
C07305=1153.669,9.241,-48.047,179.859,6.140,149.148
C07306=1153.664,9.492,-48.061,179.862,6.140,149.147
C07307=1153.658,9.741,-48.075,179.864,6.141,149.147
C07308=1153.653,9.990,-48.089,179.866,6.142,149.146
C07309=1153.649,10.240,-48.102,179.869,6.143,149.146
C07310=1153.643,10.489,-48.116,179.872,6.144,149.145
C07311=1153.638,10.739,-48.130,179.874,6.145,149.145
C07312=1153.632,10.988,-48.144,179.877,6.145,149.144
C07313=1153.628,11.238,-48.157,179.879,6.146,149.143
C07314=1153.623,11.488,-48.171,179.881,6.146,149.143
C07315=1153.617,11.737,-48.185,179.884,6.148,149.142
C07316=1153.612,11.987,-48.199,179.887,6.148,149.142
C07317=1153.607,12.237,-48.213,179.889,6.149,149.141
C07318=1153.602,12.485,-48.226,179.892,6.150,149.140
C07319=1153.597,12.735,-48.241,179.894,6.151,149.140
C07320=1153.592,12.986,-48.254,179.897,6.152,149.139
C07321=1153.587,13.235,-48.268,179.899,6.153,149.139
C07322=1153.582,13.484,-48.283,179.902,6.153,149.138
C07323=1153.577,13.734,-48.297,179.904,6.154,149.138
C07324=1153.572,13.983,-48.310,179.907,6.155,149.137
C07325=1153.567,14.233,-48.324,179.910,6.156,149.137
